// §7.6.1 — single gated manual-command entry for the HMI. Accepts ONLY when this
// Unit is in MANUAL (§3.4) AND the user holds MANUAL access (§7.7). Routes to the
// target module's ManualCommand (through the command surface — defended, not
// bypassed). Logs every accept/reject as a §8.3 event. Concrete Units override
// _M_RouteManual to map TargetPath -> the child module.
METHOD ManualCommandTo : BOOL
VAR_INPUT
    TargetPath : STRING(255);
    Value : DINT;
END_VAR
VAR
    auditSlot : INT;
END_VAR
ManualCommandTo := FALSE;
IF _mode <> E_Mode.MANUAL THEN
    auditSlot := AlarmLog.Raise(Reason := E_Reason.NONE,
        Text := 'std.audit.manualCommandWrongMode', Source := TargetPath,
        Severity := E_Severity.LOW, Category := E_Category.SYSTEM, ResetClass := E_ResetClass.AUTO_RESET);
    IF auditSlot > 0 THEN AlarmLog.Gone(Slot := auditSlot); END_IF
    RETURN;
END_IF
IF NOT Access.PermitsLogged(Gate := E_GatedAction.MANUAL) THEN
    RETURN;                              // §7.7 denial already audited
END_IF
ManualCommandTo := _M_RouteManual(TargetPath := TargetPath, Value := Value);
IF ManualCommandTo THEN
    auditSlot := AlarmLog.Raise(Reason := E_Reason.NONE,
        Text := 'std.audit.manualCommandAccepted', Source := TargetPath,
        Severity := E_Severity.LOW, Category := E_Category.SYSTEM, ResetClass := E_ResetClass.AUTO_RESET);
ELSE
    auditSlot := AlarmLog.Raise(Reason := E_Reason.UNSUPPORTED_COMMAND,
        Text := 'std.audit.manualCommandRejected', Source := TargetPath,
        Severity := E_Severity.LOW, Category := E_Category.SYSTEM, ResetClass := E_ResetClass.AUTO_RESET);
END_IF
IF auditSlot > 0 THEN AlarmLog.Gone(Slot := auditSlot); END_IF
END_METHOD

PROPERTY ModeActive : E_Mode
GET
ModeActive := _mode;
END_GET
END_PROPERTY

PROPERTY ModelCode : STRING(64)
GET
ModelCode := Model.ModelCode;
END_GET
END_PROPERTY

PROPERTY ModuleType : E_ModuleType
GET
ModuleType := E_ModuleType.UNIT;
END_GET
END_PROPERTY

// base first (§3.14.2); then children, one-shot init, mode transition, stall watch
METHOD PROTECTED OnCyclic : DINT
VAR
    publishIdx : INT;
    modeIdx    : E_Mode;
    styleIdx   : E_RunStyle;
    previousMode : E_Mode;
    modeExitResult : DINT;
    highestSeverity : E_Severity;
    alarmActive : BOOL;
    heldReported : BOOL;
END_VAR
OnCyclic := SUPER^.OnCyclic();
_M_SyncModelCatalog();
_M_BeginSequenceScan();                               // §6.10 one-scan result reset for every attached chain
_M_TickChildren();
IF _pLine <> 0 THEN
    IF _lineHost THEN
        _pLine^.Cyclic();                             // §3.8e the hosting root runs the line
    END_IF
    // A line value can change without a write through THIS root: a mirror applies
    // its owner's revision, a second root on the line edits it. Either way this
    // root's manifest now reads differently, so its revision moves.
    IF _pLine^.OutImm.Revision <> _lineRevSeen THEN
        _lineRevSeen := _pLine^.OutImm.Revision;
        ConfigRev := ConfigRev + 1;
    END_IF
END_IF
_M_OeeUpdate();                                       // §8.5.1 time accounting + sampling
M_ShiftTick(Now := F_Now(), Synchronized := F_TimeSynchronized());   // §8.5.2
AlarmLog.Cyclic();                                    // §8.10 shelf auto-expiry
_M_EngineeringCyclic();                               // §7.5.2 standing gate annunciation
_healthPublisher.Cyclic(Input := _healthInput, ParCfg := _healthParCfg,
    Configured := _healthConfigured);                 // §2.7/§8.12 alarm edges + values
SystemHealth := _healthPublisher.Status;
_M_ChartRevCyclic();                                  // §3.13 coalesced chart revision
_M_HeldCyclic();                                      // §7.6.1a hold-to-run re-assert
_M_ConfigPersistCyclic();                             // §3.8b durability window
_M_DrainRestoreLoss();                                // §3.8b restore annunciation
_M_HandleHmiRequest();                                // §3.10 request mailbox
_M_DecisionCyclic();                                  // §6.11 timeout/default/overlap resolver
Access.Cyclic();
alarmActive := _M_HighestSeverity(Highest := highestSeverity);
_towerMapper.Cyclic(MachineState := MachineState, AlarmActive := alarmActive,
    HighestSeverity := highestSeverity,
    OperatorActionRequired := (Decision.Prompt <> ''),
    LampTestRequest := _lampTestRequest, ParCfg := _towerParCfg);
_lampTestRequest := FALSE;
SignalTower := _towerMapper.Status;
// §9.8 data-driven Control On/Off request endpoint. Off wins if both arrive;
// the domain/power-group implementation still validates safety, health and rearm.
ControlOnRequest := FALSE;
ControlOffRequest := FALSE;
IF ReqControlOff THEN
    ReqControlOff := FALSE;
    ReqControlOn := FALSE;
    IF Access.PermitsLogged(Gate := E_GatedAction.POWER_CONTROL) THEN
        ControlOffRequest := TRUE;
    END_IF
ELSIF ReqControlOn THEN
    ReqControlOn := FALSE;
    IF Access.PermitsLogged(Gate := E_GatedAction.POWER_CONTROL) THEN
        ControlOnRequest := TRUE;
    END_IF
END_IF
// §3.14.4 — pending mode change; §3.4.1 style decides graceful vs immediate
IF _modePend THEN
    IF _exec = E_ExecState.BUSY THEN
        IF ModePolicy[TO_INT(_mode)].Style = E_ModeSwitchStyle.GRACEFUL THEN
            _stopReq := TRUE;                             // finish the cycle at its stop point
        ELSE
            modeExitResult := OnModeExit(FirstCall := _modeExitFirst,
                RequestedMode := _modeReq);
            _modeExitFirst := FALSE;
            IF modeExitResult = 0 THEN
                OnAbort();                                // IMMEDIATE: cancel now (override may defer)
            END_IF
        END_IF
    ELSE
        IF _exec <> E_ExecState.READY THEN
            Execute := FALSE;                             // release the run command (§6.1 reset)
        ELSE
            previousMode := _mode;
            _mode := _modeReq;
            _modePend := FALSE;
            _modeExitFirst := FALSE;
            _M_CascadeMode(_mode);                        // §3.7 cascade [TC3]
            OnModeChanged(NewMode := _mode, OldMode := previousMode);
        END_IF
    END_IF
END_IF
// §8.3(c) — automatic fault capture: ERROR entry raises, ERROR exit marks gone
IF (_exec = E_ExecState.ERROR) AND (_faultEvt = 0) THEN
    _faultEvt := AlarmLog.RaiseDiag(D := _diag, ResetClass := E_ResetClass.MANUAL_RESET);
    _M_PartAborted();                  // §3.16.3: a faulted part leaves without a valid result
ELSIF (_exec <> E_ExecState.ERROR) AND (_faultEvt > 0) THEN
    AlarmLog.Gone(Slot := _faultEvt);                            // -> WAIT_RESET (blocking)
    _faultEvt := 0;
END_IF
// §6.9 — instant rollup on awaited Error; adopt a HELD child; stall as PENDING otherwise
IF _exec = E_ExecState.BUSY THEN
    IF (_awaits <> 0) AND_THEN _awaits.FaultActive THEN
        _M_FaultDiag(_awaits.GetFaultSummary());
    ELSE
        // §6.1 HELD — the held module is waiting on a condition it can name, so
        // report THAT instead of letting StallTime expire into a generic stall. A
        // declared wait is not a stall, so the watchdog stays disarmed while it lasts.
        //
        // The hold rolls up whether or not the step awaits the child (§1.1 O1: the
        // project must not have to remember a call to stay correct). `Awaits := 0`
        // says "this step owns the child's FAULT disposition" (§6.9, press AUTO
        // N200 offering scrap/return) - it does not say "stay silent while the ram
        // is HELD". A hold is recoverable information that clears itself and never
        // blocks a restart, so suppressing it only produced a Unit that sat BUSY
        // with an empty diagnostic while its own child correctly reported Held.
        // Prefer the awaited module: when a step named one it is the most specific
        // source. _M_RollupHold is called on exactly the scans the awaited branch
        // did not fire, because TwinCAT does not short-circuit and calling both
        // would let a second held child overwrite the named one.
        heldReported := FALSE;
        IF (_awaits <> 0) AND_THEN _awaits.HoldActive THEN
            _M_HoldDiag(Diag := _awaits.GetFaultSummary());
            heldReported := TRUE;
        ELSE
            heldReported := _M_RollupHold();   // §8.2 first held registered child
        END_IF
        IF heldReported THEN
            _tStall(IN := FALSE);
        ELSE
            IF Held THEN
                _M_ClearPending();     // the hold ended: drop any stall text it outlived
            END_IF
            _tStall(IN := TRUE, PT := SEL(CurrentStep.ExpectedTime > T#0S, StallTime, CurrentStep.ExpectedTime));
            IF _tStall.Q THEN
                _M_StallWalk();
            END_IF
        END_IF
    END_IF
ELSE
    _tStall(IN := FALSE);
END_IF
// §6.9(a) — every new fault joins the shift-change ring, no historian needed
_fTrig(CLK := (_exec = E_ExecState.ERROR));
_errClr(CLK := (_exec <> E_ExecState.ERROR));
IF _errClr.Q THEN
    _M_ResumeSequencesAfterError();   // §6.9 re-evaluate, do not resume blind
END_IF
IF _fTrig.Q THEN
    _M_PushHistory(_diag);
END_IF
// §8.11.4(d) — creeping WORK time is a MAINTENANCE event (Low), not downtime:
// the profiler pulses once per excursion past the configured baseline band.
IF Profiler.DegradedTrig THEN
    _M_RaiseMaintenance(Reason := E_Reason.CYCLE_TIME_DEGRADED,
        Text := 'std.maintenance.cycleTimeDegraded');
END_IF
ModeActivePublished := _mode;
RunningPublished := (_exec = E_ExecState.BUSY);
StopPendingPublished := _stopReq AND (_exec = E_ExecState.BUSY);
FOR publishIdx := 0 TO PL_Fraktal.MODE_COUNT - 1 DO
    modeIdx := publishIdx;
    SupportedModesPublished[publishIdx] := _M_Supports(Mode := modeIdx);
END_FOR
FOR publishIdx := 0 TO 2 DO
    styleIdx := publishIdx;
    SupportedRunStylesPublished[publishIdx] := _M_SupportsRunStyle(Style := styleIdx);
END_FOR
END_METHOD

// §8.13 — derive the tower input from the authoritative active-event table.
METHOD PRIVATE _M_HighestSeverity : BOOL
VAR_IN_OUT
    Highest : E_Severity;
END_VAR
VAR
    i : INT;
END_VAR
_M_HighestSeverity := FALSE;
Highest := E_Severity.LOW;
FOR i := 1 TO PL_Fraktal.MAX_ALARM_ACTIVE DO
    IF AlarmLog.Active[i].State <> E_AlarmState.CLOSED THEN
        IF NOT _M_HighestSeverity OR (AlarmLog.Active[i].Severity > Highest) THEN
            Highest := AlarmLog.Active[i].Severity;
        ELSE
            ;
        END_IF
        _M_HighestSeverity := TRUE;
    ELSE
        ;
    END_IF
END_FOR
END_METHOD

// §8.13 — remote request is MANUAL-gated and starts only while the Unit is idle.
METHOD RequestLampTest : BOOL
RequestLampTest := FALSE;
IF _exec = E_ExecState.BUSY THEN
    RETURN;
END_IF
IF NOT Access.PermitsLogged(Gate := E_GatedAction.MANUAL) THEN
    RETURN;
END_IF
_lampTestRequest := TRUE;
RequestLampTest := TRUE;
END_METHOD

// Startup station-convention seam. Runtime config writes require a registered
// typed capability; this method is not published by OPC UA.
METHOD SetSignalTowerConfig : BOOL
VAR_INPUT
    ParCfg : ST_SignalTowerParCfg;
END_VAR
IF (ParCfg.SchemaVersion <> 1) OR (ParCfg.LampTestDuration <= T#0S) THEN
    SetSignalTowerConfig := FALSE;
    RETURN;
END_IF
_towerParCfg := ParCfg;
SetSignalTowerConfig := TRUE;
END_METHOD

// TC3/platform adapter injection. Raw probe values remain OPC-UA-hidden; the
// health publisher validates and republishes the bounded status surface.
METHOD SetSystemHealth : BOOL
VAR_INPUT
    Input  : ST_SystemHealthInput;
    ParCfg : ST_SystemHealthParCfg;
END_VAR
IF ParCfg.SchemaVersion <> 1 THEN
    SetSystemHealth := FALSE;
    RETURN;
END_IF
_healthInput := Input;
_healthParCfg := ParCfg;
_healthConfigured := TRUE;
SetSystemHealth := TRUE;
END_METHOD

// §3.14 hook — one-shot after first operational scan
METHOD PROTECTED OnInit : DINT
VAR
    i : INT;
END_VAR
OnInit := SUPER^.OnInit();
_M_RestartSequences();         // §6.8 every attached chain starts at N000
SequenceViewEnabled := TRUE;   // §3.13 a Unit has a chain worth drawing;
                               // a concrete Unit may vary this per mode
Access.Setup(Provider := 0, pAlarmLog := ADR(AlarmLog)); // preserves an injected provider
_healthPublisher.Setup(SourcePath := CONCAT(Status.Name, '.SystemHealth'),
    pAlarmLog := ADR(AlarmLog));
// §3.10.2 — seed the manifest revision from boot time so every PLC restart or
// re-activation yields a NEW value (a plain counter would repeat after reboot
// and an HMI could keep a stale manifest undetected). Config writes increment.
ConfigRev := DT_TO_UDINT(F_Now());
// §3.8b — the durability provider defaults to the shipped LOCAL_RETAIN writer.
// SetConfigPersistence may already have replaced it, so this never overwrites an
// injected one.
IF _persistence = 0 THEN
    _persistence := _persistWriter;
END_IF
_liveArmed := TRUE;            // §3.8b the walk is complete: the documents may restore
// The framework's OWN station config is subject to the same rule it imposes on
// every module: version 0 is a first boot that lost nothing, any other
// unrecognized version means a real ModePolicy image was rejected and that is
// annunciated with this root's path. The base used to treat both cases as a
// silent re-initialize, which is exactly the "runs on defaults while presenting
// itself as commissioned" failure §3.8b exists to prevent.
IF NOT M_RestoreStationCfg(pVersion := ADR(_modePolicyVersion),
        SchemaVersion := MODE_POLICY_SCHEMA) THEN
    _M_InitModePolicy();
    FOR i := 0 TO PL_Fraktal.MODE_COUNT - 1 DO
        _modePolicyStored[i] := ModePolicy[i];
    END_FOR
ELSE
    FOR i := 0 TO PL_Fraktal.MODE_COUNT - 1 DO
        ModePolicy[i] := _modePolicyStored[i];
    END_FOR
END_IF
END_METHOD

// §3.14 hook — after the new mode is committed
METHOD PROTECTED OnModeChanged : DINT
VAR_INPUT
    NewMode : E_Mode;
    OldMode : E_Mode;
END_VAR
_M_HostEvent(Kind := E_HostEventKind.MODE_CHANGED, PartUid := '',
    Subject := 'Mode', Value := TO_STRING(TO_DINT(NewMode)),
    Verdict := E_Verdict.NONE, ReasonCode := E_Reason.NONE);
// §3.13 — the chart belongs to the mode that is running. A project writes nothing
// for this: it lands in the base hook every override calls SUPER^ on first (§3.14.2).
_M_ResetSequenceRows();
// §6.8 — and so do the chains: a new mode starts every chain at N000.
_M_RestartSequences();
OnModeChanged := 0;
END_METHOD

// Core §11.6: CHANGEOVER starts when its guided sequence actually starts, not
// merely when the operator selects the mode or transactionally loads a model.
METHOD PROTECTED OnCommandStart : DINT
OnCommandStart := SUPER^.OnCommandStart();
IF _mode = E_Mode.CHANGEOVER THEN
    _M_HostEvent(Kind := E_HostEventKind.CHANGEOVER_STARTED, PartUid := '',
        Subject := 'Model', Value := Model.ModelCode,
        Verdict := E_Verdict.NONE, ReasonCode := E_Reason.NONE);
END_IF
END_METHOD

// §3.14.4 — called every scan while a mode request is pending and the Unit is BUSY.
// Return 0 = consent to immediate cancel (default); >0 = still stopping gracefully.
METHOD PROTECTED OnModeExit : DINT
VAR_INPUT
    FirstCall : BOOL;
    RequestedMode : E_Mode;
END_VAR
OnModeExit := 0;
END_METHOD

// §8.3(b) — deliberate operator reset of blocking events (release-gated per §7.6/§14).
// ONE operator action has to make the Unit restartable, so this closes the blocking
// events AND clears the latched control state they were reporting: see _M_RecoverState.
METHOD OperatorReset : BOOL
IF NOT Access.PermitsLogged(Gate := E_GatedAction.ALARM_RESET) THEN
    OperatorReset := FALSE;            // §7.7
    RETURN;
END_IF
OperatorReset := _M_RecoverState();
OperatorReset := AlarmLog.OperatorReset() OR OperatorReset;
END_METHOD

// §8.3(b)/§6.1 — the control-state half of a reset. Closing the alarm alone left the
// machine locked: the Unit's run command and the child commands its mode chain had
// issued both stayed asserted, and §6.1's Execute-drop reset — the only exit from a
// latched terminal state — needs them LOW. A frozen chain cannot drop them itself,
// because a Unit that is not BUSY never calls _M_Dispatch again, so the step holding
// `child.Execute := TRUE` never runs. Nothing else in the system clears it, and the
// next Start re-issues the same already-TRUE input: no rising edge, the child stays
// in ERROR, and the Unit re-adopts the fault through the §8.2 rollup. That is the
// press hard-lock. Returns TRUE when there was something to recover.
// Deliberately does NOT clear ERROR here: Cyclic keeps that ownership (§6.1), so a
// cause that is still live re-faults on the next command edge instead of vanishing.
METHOD PROTECTED _M_RecoverState : BOOL
_M_RecoverState := FALSE;
IF (_exec <> E_ExecState.ERROR) AND NOT AlarmLog.Blocking THEN
    RETURN;                            // nothing latched: a stray reset changes nothing
END_IF
OnOperatorReset();                     // §3.14 hook: withdraw outputs, reset mode chains
_M_ReleaseChildCommands();             // stranded child commands -> READY next scan
_M_ClearPending();
_stopReq := FALSE;
IF _exec = E_ExecState.BUSY THEN
    // Defined safe reaction (§5.6) for a blocking event raised by application code
    // while the mode chain still runs: a recovery reset cancels what was running
    // rather than leaving a chain we just reset still driving the machine.
    AbortCommand();
END_IF
Execute  := FALSE;                     // stale run command -> Unit READY next scan
_faultEvt := 0;                        // the event is closed here, not by a later Gone()
_M_RecoverState := TRUE;
END_METHOD

// §3.14 hook — an accepted operator reset is recovering this Unit. Override to
// withdraw application outputs and reset application-owned mode chains before the
// base releases the run command; call SUPER^.OnOperatorReset() first (§3.14.2).
// Called only when something was actually latched (ERROR or a blocking alarm), so an
// override may assume it is a recovery, not a routine poll.
METHOD PROTECTED OnOperatorReset : DINT
OnOperatorReset := 0;
END_METHOD

// Application-only seam for an ordinary hardwired fault-reset/acknowledge button,
// mirroring RequestLocalControl (§9.8): it is a METHOD, not OPC UA data, so remote
// clients still go through the access-gated OPERATOR_RESET request and cannot reach
// this path. A cabinet button IS its own authorization (physical presence), so it
// carries no §7.7 session check — but the reset is still audited as a §8.3 event,
// and it recovers exactly the same state as an operator reset, never more.
// The composition root calls this from its hardware driver on the button's rising
// edge, once per root Unit it should clear.
METHOD RequestLocalReset : BOOL
VAR
    auditSlot : INT;
END_VAR
auditSlot := AlarmLog.Raise(Reason := E_Reason.NONE,
    Text := 'std.audit.localResetRequested', Source := _name,
    Severity := E_Severity.LOW, Category := E_Category.SYSTEM,
    ResetClass := E_ResetClass.AUTO_RESET);
IF auditSlot > 0 THEN AlarmLog.Gone(Slot := auditSlot); END_IF
RequestLocalReset := _M_RecoverState();
RequestLocalReset := AlarmLog.OperatorReset() OR RequestLocalReset;
END_METHOD

// §3.8 optional HMI/MES selection catalog. Recipe providers remain pluggable;
// the application registers only the model identities it deliberately exposes.
METHOD RegisterAvailableModel : BOOL
VAR_INPUT
    Id : ST_ModelId;
END_VAR
VAR
    i : INT;
END_VAR
RegisterAvailableModel := FALSE;
IF (Id.ModelCode = '') OR (AvailableModelCount >= PL_Fraktal.MAX_RECIPES) THEN
    RETURN;
END_IF
FOR i := 1 TO AvailableModelCount DO
    IF AvailableModels[i].ModelCode = Id.ModelCode THEN
        RETURN;
    END_IF
END_FOR
AvailableModels[AvailableModelCount + 1] := Id;
AvailableModelCount := AvailableModelCount + 1;
ConfigRev := ConfigRev + 1;    // §3.10.2 — manifest changed
RegisterAvailableModel := TRUE;
END_METHOD

// §9.8 remote control-domain request. The acknowledgement is the result of this
// authorization check; it is never reported accepted before POWER_CONTROL runs.
METHOD RequestControlPower : BOOL
VAR_INPUT
    ControlOn : BOOL;
END_VAR
RequestControlPower := FALSE;
IF NOT Access.PermitsLogged(Gate := E_GatedAction.POWER_CONTROL) THEN
    RETURN;
END_IF
IF ControlOn THEN
    ReqControlOn := TRUE;
    ReqControlOff := FALSE;
ELSE
    ReqControlOff := TRUE;                         // Off wins if both were requested
    ReqControlOn := FALSE;
END_IF
RequestControlPower := TRUE;
END_METHOD

// §6.11 authoritative decision entry. START_STOP is the access gate because the
// answer advances a running Unit chain; option-specific process releases append
// through _M_AppendDecisionInterlocks. A stale/invalid answer never latches.
METHOD SubmitDecision : BOOL
VAR_INPUT
    Option : INT;
END_VAR
VAR_IN_OUT
    Report : ST_ReleaseReport;
END_VAR
Report.Count := 0;
Report.Released := FALSE;
SubmitDecision := FALSE;
IF NOT Access.PermitsLogged(Gate := E_GatedAction.START_STOP) THEN
    _M_AddReason(Report := Report, Text := 'std.release.insufficientStartStop',
        Reason := E_Reason.NONE, Kind := E_ReleaseKind.ACCESS);
END_IF
IF (_exec <> E_ExecState.BUSY) OR (Decision.Prompt = '') THEN
    _M_AddReason(Report := Report, Text := 'std.release.noActiveDecision',
        Reason := E_Reason.NONE, Kind := E_ReleaseKind.OTHER);
ELSIF (Option < 1) OR (Option > PL_Fraktal.MAX_OPTIONS) THEN
    _M_AddReason(Report := Report, Text := 'std.release.invalidDecisionOption',
        Reason := E_Reason.UNSUPPORTED_COMMAND, Kind := E_ReleaseKind.OTHER);
ELSIF Decision.Options[Option] = '' THEN
    _M_AddReason(Report := Report, Text := 'std.release.invalidDecisionOption',
        Reason := E_Reason.UNSUPPORTED_COMMAND, Kind := E_ReleaseKind.OTHER);
ELSE
    _M_AppendDecisionInterlocks(Option := Option, Report := Report);
END_IF
Report.Released := (Report.Count = 0);
IF Report.Released THEN
    DecisionAnswer := Option;
    SubmitDecision := TRUE;
END_IF
END_METHOD

// §7.7 persistent per-root policy edit. The policy's own ACCESS_POLICY threshold
// is rechecked before any threshold — including itself — can change.
METHOD SetAccessLevel : BOOL
VAR_INPUT
    Gate : E_GatedAction;
    Level : E_AccessLevel;
END_VAR
SetAccessLevel := FALSE;
IF NOT Access.PermitsLogged(Gate := E_GatedAction.ACCESS_POLICY) THEN
    RETURN;
END_IF
// Never allow an anonymous/lower session to raise the policy above itself and
// strand the retained station configuration without a usable administrator.
IF (Gate = E_GatedAction.ACCESS_POLICY) AND (Level > Access.CurrentLevel) THEN
    RETURN;
END_IF
SetAccessLevel := Access.ConfigureRequired(Gate := Gate, Level := Level);
IF SetAccessLevel THEN
    ConfigRev := ConfigRev + 1;
END_IF
END_METHOD

// §7.7 persistent idle timeout (0 = never), self-gated by ACCESS_POLICY.
METHOD SetSessionTimeout : BOOL
VAR_INPUT
    TimeoutMs : UDINT;
END_VAR
SetSessionTimeout := FALSE;
IF NOT Access.PermitsLogged(Gate := E_GatedAction.ACCESS_POLICY) THEN
    RETURN;
END_IF
SetSessionTimeout := Access.ConfigureSessionTimeout(TimeoutMs := TimeoutMs);
IF SetSessionTimeout THEN
    ConfigRev := ConfigRev + 1;
END_IF
END_METHOD

// §3.8a/§7.7 centralized HMI configuration authority. Concrete overrides never
// need to remember DATA_WRITE or root ownership; they validate only their field.
METHOD WriteConfig : BOOL
VAR_INPUT
    TargetPath : STRING(255);
    WriteKey : STRING(160);
    Revision : DINT;
    TextValue : STRING(255);
END_VAR
WriteConfig := FALSE;
IF NOT _M_ConfigRestored() THEN
    RETURN;                            // §3.8b the restore would replay over it
END_IF
IF (WriteKey = '') OR (Revision <= 0)
OR NOT _M_OwnsModulePath(Path := TargetPath) THEN
    RETURN;
END_IF
// §3.8d - the VALUE's effective write level (its class, raised by its own
// minimum); DATA_WRITE for a value in the built-in class, as before.
IF NOT Access.M_PermitsLevelLogged(Required := _M_DataLevelOf(TargetPath := TargetPath,
        WriteKey := WriteKey, ForWrite := TRUE)) THEN
    RETURN;
END_IF
WriteConfig := _M_WriteBaseConfig(TargetPath := TargetPath, WriteKey := WriteKey,
    Revision := TO_UDINT(Revision), TextValue := TextValue, Commit := TRUE);
IF NOT WriteConfig THEN
    WriteConfig := _M_RouteConfigWrite(TargetPath := TargetPath,
        WriteKey := WriteKey, Revision := TO_UDINT(Revision), TextValue := TextValue);
END_IF
// §3.8a - a model-data value lives in a recipe record too. Another model's edit
// exists ONLY in that record, so failing to save it fails the write; the active
// model's edit is already live, and saving it keeps it across a changeover.
IF WriteConfig AND (TargetPath = Status.Name) AND _M_ModelScopedKey(WriteKey := WriteKey) THEN
    IF NOT _M_SaveModelData() AND (_pModelView <> 0) THEN
        WriteConfig := FALSE;
    END_IF
END_IF
IF WriteConfig THEN
    ConfigRev := ConfigRev + 1;
    _M_MarkPersistPending();           // §3.8b: accepted is LIVE, not yet DURABLE
END_IF
END_METHOD

// §3.8c - the root authority for a capture. Deliberately the same gate, the same
// ownership check and the same ConfigRev bump as WriteConfig: a capture is a
// write whose value came from the machine, and it is no more and no less
// privileged than one the operator typed (§3.8c(d)).
METHOD CaptureConfig : BOOL
VAR_INPUT
    TargetPath : STRING(255);
    WriteKey   : STRING(160);
    Revision   : DINT;
END_VAR
CaptureConfig := FALSE;
IF NOT _M_ConfigRestored() THEN
    RETURN;
END_IF
IF (WriteKey = '') OR (Revision <= 0)
OR NOT _M_OwnsModulePath(Path := TargetPath) THEN
    RETURN;
END_IF
IF NOT Access.M_PermitsLevelLogged(Required := _M_DataLevelOf(TargetPath := TargetPath,
        WriteKey := WriteKey, ForWrite := TRUE)) THEN
    RETURN;
END_IF
// Framework-owned keys offer no capture: they are policy, not measurements.
CaptureConfig := M_ApplyCapture(Scope := TargetPath, WriteKey := WriteKey,
    Revision := TO_UDINT(Revision), RootReady := (_exec = E_ExecState.READY));
IF CaptureConfig THEN
    ConfigRev := ConfigRev + 1;
END_IF
END_METHOD

// Core §7.5.1 — inject the station's commissioning/engineering gate register at
// Setup, the same shape as SetPartCarrier. Wiring it is what makes the §7.5.2
// standing annunciation appear and what arms the §10.5.1 force surface; a Unit
// with no register is a production Unit and both are simply absent.
//
// Declaring the framework's OWN force gate happens here rather than in the
// project, so a composition root that wires the register cannot forget it
// (§1.1 O1) and cannot arm forcing without also annunciating it.
METHOD SetEngineeringMode
VAR_INPUT
    Mode : REFERENCE TO FB_EngineeringMode;
END_VAR
_engineering REF= Mode;
IF __ISVALIDREF(_engineering) THEN
    _engineering.M_DeclareOutputForcing();
ELSE
    ;
END_IF
END_METHOD

// Core §10.5.1 rules 1 and 3 — may a held force set-point be applied to this
// Unit's outputs right now? The project hardware driver passes the result to
// FB_IoTopologyPublisher.M_ApplyForces every scan, and ForceChannel gates the
// operator request on the identical predicate, so "accepted" and "applied" can
// never disagree. Everything else about a force (access, ownership, direction,
// mapping) is proved elsewhere; this is only the build gate and the mode/state.
METHOD M_ForcePermitted : BOOL
M_ForcePermitted := FALSE;
IF NOT __ISVALIDREF(_engineering) THEN
    RETURN;
END_IF
IF NOT _engineering.ForcingActive THEN
    RETURN;
END_IF
// A running module reasserts its own outputs, so a force is only honest while
// the Unit is idle in MANUAL; leaving either withdraws every force (§10.5.1(3)).
M_ForcePermitted := (_mode = E_Mode.MANUAL) AND (_exec = E_ExecState.READY);
END_METHOD

// Core §7.5.2 — the standing annunciation: one LOW/SYSTEM/AUTO_RESET event per
// registered gate, for as long as that gate is registered.
//
// Why each choice is the way it is, because every one of them is load-bearing:
//   AUTO_RESET  a MANUAL_RESET event refuses Start (§8.3(b)), which would make
//               commissioning gates block the commissioning they exist to serve;
//   LOW/SYSTEM  the lowest priority and the lowest risk class - this says how the
//               software was BUILT, not that the process or safety is impaired,
//               and a louder class would displace real alarms (§8.9);
//   unclearable OperatorReset only closes MANUAL_RESET events, so no operator
//               action reaches this one, and its §8.9 record is not shelvable, so
//               §8.10 cannot silence it either. It closes when the gate is gone -
//               which, gates being build constants, means a new download.
METHOD PRIVATE _M_EngineeringCyclic
VAR
    i : INT;
    gateCount : INT;
END_VAR
IF NOT __ISVALIDREF(_engineering) THEN
    RETURN;
END_IF
gateCount := _engineering.Count;
IF gateCount > PL_Fraktal.MAX_ENGINEERING_GATES THEN
    gateCount := PL_Fraktal.MAX_ENGINEERING_GATES;
END_IF
FOR i := 1 TO gateCount DO
    // Self-healing on purpose. If this slot were ever closed and reused by
    // another event, a remembered index would leave the annunciation silently
    // absent for the rest of the run - the one failure mode a non-clearable
    // message must not have. Re-verify identity, then re-raise.
    IF _engineeringEvt[i] > 0 THEN
        IF (AlarmLog.Active[_engineeringEvt[i]].State = E_AlarmState.CLOSED)
        OR (AlarmLog.Active[_engineeringEvt[i]].ReasonCode <> E_Reason.COMMISSIONING_GATE_ACTIVE) THEN
            _engineeringEvt[i] := 0;
        ELSE
            ;
        END_IF
    ELSE
        ;
    END_IF
    IF _engineeringEvt[i] = 0 THEN
        _engineeringEvt[i] := AlarmLog.Raise(Reason := E_Reason.COMMISSIONING_GATE_ACTIVE,
            Text := _engineering.Gates[i].DescriptionKey, Source := _name,
            Severity := E_Severity.LOW, Category := E_Category.SYSTEM,
            ResetClass := E_ResetClass.AUTO_RESET);
    ELSE
        ;
    END_IF
END_FOR
END_METHOD

// §10.5.1 centralized force authority. Only an idle MANUAL Unit may reach the
// application resolver; that resolver still proves root ownership, OUTPUT,
// non-safety identity, mapping and the channel-specific release.
METHOD ForceChannel : BOOL
VAR_INPUT
    ChannelPath : STRING(255);
    Force : BOOL;
    BoolText : STRING(255);
    AnalogText : STRING(160);
END_VAR
ForceChannel := FALSE;
IF NOT Access.PermitsLogged(Gate := E_GatedAction.MANUAL) THEN
    RETURN;
END_IF
// §10.5.1 rules 1 and 3 in one predicate, the same one the hardware driver
// applies each scan - so the request can never be accepted under conditions
// under which the force would not actually be applied.
IF NOT M_ForcePermitted() OR (ChannelPath = '') THEN
    RETURN;
END_IF
ForceChannel := _M_RouteForceChannel(ChannelPath := ChannelPath, Force := Force,
    BoolText := BoolText, AnalogText := AnalogText);
END_METHOD

// Core §7.8 — full rollup for the simpler gated Unit actions (Stop, ALARM_RESET,
// CHANGEOVER, MODE_CHANGE, step). Same predicate the gates use. Start has its own
// richer ReleaseReportStart (interlocks); manual has ReleaseReportManual (target).
METHOD ReleaseReportAction : BOOL
VAR_INPUT
    Gate : E_GatedAction;
END_VAR
VAR_IN_OUT
    Report : ST_ReleaseReport;
END_VAR
Report.Count := 0;
Report.Released := FALSE;
// access is the common gate
IF NOT Access.Permits(Gate := Gate) THEN
    _M_AddReason(Report := Report, Text := 'std.release.insufficientAction', Reason := E_Reason.NONE, Kind := E_ReleaseKind.ACCESS);
END_IF
// per-action state preconditions
CASE Gate OF
    E_GatedAction.CHANGEOVER:
        IF _exec = E_ExecState.BUSY THEN
            _M_AddReason(Report := Report, Text := 'std.release.changeoverRunning', Reason := E_Reason.NONE, Kind := E_ReleaseKind.MODE);
        END_IF
    E_GatedAction.ALARM_RESET:
        IF NOT AlarmLog.Blocking THEN
            _M_AddReason(Report := Report, Text := 'std.release.noBlockingAlarm', Reason := E_Reason.NONE, Kind := E_ReleaseKind.OTHER);
        END_IF
    E_GatedAction.MODE_CHANGE:
        IF _modePend THEN
            _M_AddReason(Report := Report, Text := 'std.release.modeChangeAlreadyPending', Reason := E_Reason.NONE, Kind := E_ReleaseKind.MODE);
        ELSIF (_exec = E_ExecState.BUSY)
        AND (ModePolicy[TO_INT(_mode)].Shield = E_ModeSwitchShield.BLOCKED_WHILE_RUNNING) THEN
            _M_AddReason(Report := Report, Text := 'std.release.modeSwitchBlockedWhileRunning',
                Reason := E_Reason.NONE, Kind := E_ReleaseKind.MODE);
        ELSE
            ;
        END_IF
ELSE
    ;                                          // actions with no extra state predicate
END_CASE
Report.Released := (Report.Count = 0);
ReleaseReportAction := Report.Released;
END_METHOD

// Core §7.8 — full rollup of why a manual command to Target would be refused (§7.6.1).
METHOD ReleaseReportManual : BOOL
VAR_INPUT
    TargetPath : STRING(255);
    Value : DINT;
END_VAR
VAR_IN_OUT
    Report : ST_ReleaseReport;
END_VAR
Report.Count := 0;
Report.Released := FALSE;
IF _mode <> E_Mode.MANUAL THEN
    _M_AddReason(Report := Report, Text := 'std.release.manualModeRequired', Reason := E_Reason.NONE, Kind := E_ReleaseKind.MODE);
END_IF
IF NOT Access.Permits(Gate := E_GatedAction.MANUAL) THEN
    _M_AddReason(Report := Report, Text := 'std.release.insufficientManual', Reason := E_Reason.NONE, Kind := E_ReleaseKind.ACCESS);
END_IF
_M_AppendManualInterlocks(TargetPath := TargetPath, Value := Value, Report := Report);  // §7.6, target+command-aware
Report.Released := (Report.Count = 0);
ReleaseReportManual := Report.Released;
END_METHOD

// Core §7.8 — pure query: the FULL rollup of why Start would be refused right now.
// This is the authoritative machine predicate consumed by Start (no drift).
// Released = TRUE means Start proceeds. Lists mode + access + blocking-alarm,
// control-domain, and concrete mode-entry release reasons. The caller owns the
// bounded report storage; returning this large record by value can overflow a
// TwinCAT task stack when Start consumes the result.
METHOD ReleaseReportStart : BOOL
VAR_IN_OUT
    Report : ST_ReleaseReport;
END_VAR
Report.Count := 0;
Report.Released := FALSE;
// access (§7.7)
IF NOT Access.Permits(Gate := E_GatedAction.START_STOP) THEN
    _M_AddReason(Report := Report, Text := 'std.release.insufficientStartStop', Reason := E_Reason.NONE, Kind := E_ReleaseKind.ACCESS);
END_IF
// mode / run state (§3.4)
IF _modePend THEN
    _M_AddReason(Report := Report, Text := 'std.release.modeChangePending', Reason := E_Reason.NONE, Kind := E_ReleaseKind.MODE);
END_IF
IF _mode = E_Mode.MANUAL THEN
    _M_AddReason(Report := Report, Text := 'std.release.manualHasNoAutoSequence', Reason := E_Reason.NONE, Kind := E_ReleaseKind.MODE);
END_IF
IF _exec <> E_ExecState.READY THEN
    _M_AddReason(Report := Report, Text := 'std.release.unitNotReady', Reason := E_Reason.NONE, Kind := E_ReleaseKind.MODE);
END_IF
// blocking alarm (§8.3)
IF AlarmLog.Blocking THEN
    _M_AddReason(Report := Report, Text := 'std.release.manualReset', Reason := E_Reason.NONE, Kind := E_ReleaseKind.ALARM);
END_IF
// lost configuration image (§3.8b): the DEPLOYMENT's declared consequence. The
// policy was stored and published but read nowhere, so a station that declared
// BLOCK_UNTIL_ACKNOWLEDGED started on defaults anyway. This is where it is read.
IF ConfigPersist.RestoreLost AND NOT ConfigPersist.RestoreAcknowledged
AND (ConfigPersist.RestorePolicy = E_ConfigRestorePolicy.BLOCK_UNTIL_ACKNOWLEDGED) THEN
    _M_AddReason(Report := Report, Text := 'std.release.configRestoreUnacknowledged', Reason := E_Reason.CONFIG_RESTORE_LOST, Kind := E_ReleaseKind.ALARM);
END_IF
// §3.8b - the live documents are still being read back: the running values are
// not yet the ones last made durable.
IF NOT _M_ConfigRestored() THEN
    _M_AddReason(Report := Report, Text := 'std.release.configRestoring', Reason := E_Reason.NONE, Kind := E_ReleaseKind.OTHER);
END_IF
IF ControlDomain.Present AND NOT ControlDomain.ReadyForStart THEN
    _M_AddReason(Report := Report, Text := 'std.release.controlDomainNotReady', Reason := E_Reason.NONE, Kind := E_ReleaseKind.INTERLOCK);
END_IF
// active mode's immediate entry/frontier conditions (concrete override)
_M_AppendInterlocks(Report := Report);
Report.Released := (Report.Count = 0);
ReleaseReportStart := Report.Released;
END_METHOD

// §8.5.1 — clear accumulators + ring (shift start). Gated: §7.7 DATA_WRITE; audited §8.3.
METHOD ResetOee : BOOL
VAR
    i : INT;
    auditSlot : INT;
END_VAR
IF NOT Access.PermitsLogged(Gate := E_GatedAction.DATA_WRITE) THEN
    ResetOee := FALSE;
    RETURN;
END_IF
_oeeGoodBase := GoodCount;
_oeeNokBase := NokCount;
Oee.RunMs := 0; Oee.DownMs := 0; Oee.IdleMs := 0;
FOR i := 1 TO PL_Fraktal.MAX_OEE_SAMPLES DO
    OeeTrend[i].Oee := 0.0; OeeTrend[i].OeeValid := FALSE;
    OeeTrend[i].Availability := 0.0; OeeTrend[i].Performance := 0.0; OeeTrend[i].Quality := 0.0;
END_FOR
OeeTrendHead := 0;
_oeeSampMs := 0;
_M_OeeCompute();
_shiftManualReset := TRUE;                  // §8.5.2(c): the shift record will say so
auditSlot := AlarmLog.Raise(Reason := E_Reason.NONE,
    Text := 'std.audit.oeeReset', Source := _name,
    Severity := E_Severity.LOW, Category := E_Category.SYSTEM, ResetClass := E_ResetClass.AUTO_RESET);
IF auditSlot > 0 THEN AlarmLog.Gone(Slot := auditSlot); END_IF
ResetOee := TRUE;
END_METHOD

// §3.4.2 — HMI HOLD_TO_RUN input. NON-SAFETY (§9): never a dead-man; interlocks
// still apply at every step. TRUE only while the operator holds the button.
METHOD SetHoldRun : BOOL
VAR_INPUT
    Held : BOOL;
END_VAR
IF Held AND (NOT Access.PermitsLogged(Gate := E_GatedAction.START_STOP)
OR (RunStyle <> E_RunStyle.HOLD_TO_RUN) OR (_exec <> E_ExecState.BUSY)) THEN
    SetHoldRun := FALSE;
    RETURN;
END_IF
_holdRun := Held;                     // FALSE is always accepted so a hold cannot stick
SetHoldRun := TRUE;
END_METHOD

// §8.5.1 — configure the ideal cycle time (per model, §3.8). 0 disables Performance.
METHOD SetIdealCycle : BOOL
VAR_INPUT
    Ms : UDINT;
END_VAR
Oee.IdealCycleMs := Ms;
SetIdealCycle := TRUE;
END_METHOD

// §3.4/§3.7 — FALSE = unsupported (graceful rejection); TRUE = committed or pending
METHOD SetMode : BOOL
VAR_INPUT
    Mode : E_Mode;
END_VAR
IF NOT Access.PermitsLogged(Gate := E_GatedAction.MODE_CHANGE) THEN
    SetMode := FALSE;                  // §7.7(c): who-gate ANDs the machine gates
    RETURN;
END_IF
IF NOT _M_Supports(Mode) THEN
    SetMode := FALSE;
    RETURN;
END_IF
IF (Mode = _mode) AND NOT _modePend THEN
    SetMode := TRUE;
    RETURN;
END_IF
// §3.4.1 shield: policy of the mode being LEFT governs while its sequence runs
IF (_exec = E_ExecState.BUSY)
AND (ModePolicy[TO_INT(_mode)].Shield = E_ModeSwitchShield.BLOCKED_WHILE_RUNNING) THEN
    SetMode := FALSE;                  // must Stop first (graceful rejection, not a fault)
    RETURN;
END_IF
IF (NOT _modePend) OR (_modeReq <> Mode) THEN
    _modeExitFirst := TRUE;
END_IF
_modeReq := Mode;
_modePend := TRUE;
SetMode := TRUE;
END_METHOD

// §3.1b/§3.8 — transactional model change: prepare the whole subtree, then commit.
METHOD SetModel : BOOL
VAR_INPUT
    Id : ST_ModelId;
END_VAR
IF NOT Access.PermitsLogged(Gate := E_GatedAction.CHANGEOVER) THEN
    SetModel := FALSE;                 // §7.7
    RETURN;
END_IF
IF _exec = E_ExecState.BUSY THEN
    SetModel := FALSE;                 // changeover is not mid-cycle (§3.8 loads at CHANGEOVER)
    RETURN;
END_IF
IF NOT PrepareRecipe(Model := Id) THEN
    AbortRecipe();
    SetModel := FALSE;
    RETURN;
END_IF
CommitRecipe();                         // infallible after successful preparation
Model := Id;                           // identity changes only after subtree commit
ConfigRev := ConfigRev + 1;            // §3.10.2 — recipe/config leaves changed
SetModel := TRUE;
END_METHOD

// §11.6.1 internal composition seam; not a remote command surface.
METHOD M_PublishMaterialChanged : BOOL
VAR_INPUT
    Material : STRING(80);
    Value    : STRING(80);
END_VAR
M_PublishMaterialChanged := _M_HostEvent(
    Kind := E_HostEventKind.MATERIAL_CHANGED, PartUid := '', Subject := Material,
    Value := Value, Verdict := E_Verdict.NONE, ReasonCode := E_Reason.NONE);
END_METHOD

// §11.6.1 internal composition seam; not a remote command surface.
METHOD M_PublishToolChanged : BOOL
VAR_INPUT
    Tool  : STRING(80);
    Value : STRING(80);
END_VAR
M_PublishToolChanged := _M_HostEvent(
    Kind := E_HostEventKind.TOOL_CHANGED, PartUid := '', Subject := Tool,
    Value := Value, Verdict := E_Verdict.NONE, ReasonCode := E_Reason.NONE);
END_METHOD

// §11.6.2 inject an optional OPC UA/MES/REST/MQTT delivery adapter.
METHOD M_SetHostEventSink : BOOL
VAR_INPUT
    Sink : I_HostEventSink;
END_VAR
M_SetHostEventSink := HostEvents.SetSink(Sink := Sink);
END_METHOD

// §3.16.2 — inject the part carrier at the composition root (0 = traceability off).
// Source-agnostic: BY_POSITION local, RFID, DataMatrix, or host, behind I_PartCarrier.
METHOD SetPartCarrier : BOOL
VAR_INPUT
    Carrier : I_PartCarrier;
END_VAR
_carrier := Carrier;
SetPartCarrier := (Carrier <> 0);
END_METHOD

// §3.4.2 — HMI selects the run style for the active mode. Modes that don't opt in
// (see _M_SupportsRunStyle) reject non-CONTINUOUS. Access: MODE_CHANGE-gated (§7.7).
METHOD SetRunStyle : BOOL
VAR_INPUT
    Style : E_RunStyle;
END_VAR
IF NOT Access.PermitsLogged(Gate := E_GatedAction.MODE_CHANGE) THEN
    SetRunStyle := FALSE;
    RETURN;
END_IF
IF (Style <> E_RunStyle.CONTINUOUS) AND NOT _M_SupportsRunStyle(Style := Style) THEN
    SetRunStyle := FALSE;               // mode didn't opt into stepping (graceful reject)
    RETURN;
END_IF
RunStyle := Style;
SetRunStyle := TRUE;
END_METHOD

// §8.10 — gated HMI entry: shelve an active alarm's ANNUNCIATION (control untouched).
// §7.7 ALARM_SHELVE + audit; refuses SAFETY / unrationalized reasons (AlarmLog rules).
METHOD ShelveAlarm : BOOL
VAR_INPUT
    Slot      : INT;
    DurationS : UDINT;
END_VAR
IF NOT Access.PermitsLogged(Gate := E_GatedAction.ALARM_SHELVE) THEN
    ShelveAlarm := FALSE;
    RETURN;
END_IF
ShelveAlarm := AlarmLog.Shelve(Slot := Slot, DurationS := DurationS);
END_METHOD

// §3.3/§6 intro — the run IS a §6.1 command.
// §7.8: ReleaseReportStart is the authoritative machine gate as well as the
// operator explanation, so a concrete Unit cannot report an interlock it ignores.
// Build directly into the published response storage: ST_ReleaseReport is too
// large for nested by-value/local copies on a small TwinCAT task stack.
METHOD Start : BOOL
IF NOT Access.PermitsLogged(Gate := E_GatedAction.START_STOP) THEN
    Start := FALSE;                    // §7.7
    RETURN;
END_IF
IF ReleaseReportStart(Report := HmiResponse.Report) THEN
    _stopReq := FALSE;                 // §8.3(b): a MANUAL_RESET event blocks restart
    Execute := TRUE;
    Start := TRUE;
ELSE
    Start := FALSE;
END_IF
END_METHOD

// §3.4.2 — HMI single-step: request advance of one step (edge-consumed by _M_StepGate).
METHOD StepRequest : BOOL
IF NOT Access.PermitsLogged(Gate := E_GatedAction.START_STOP)
OR (RunStyle <> E_RunStyle.SINGLE_STEP) OR (_exec <> E_ExecState.BUSY) THEN
    StepRequest := FALSE;
    RETURN;
END_IF
_stepReq := TRUE;
StepRequest := TRUE;
END_METHOD

// §3.3 — stop after the current cycle
METHOD Stop : BOOL
IF NOT Access.PermitsLogged(Gate := E_GatedAction.START_STOP) THEN
    Stop := FALSE;                     // §7.7
    RETURN;
END_IF
IF _exec = E_ExecState.BUSY THEN
    _stopReq := TRUE;
ELSE
    _stopReq := FALSE;
    Execute := FALSE;                  // release a terminal run command (ERROR/DONE/ABORTED)
END_IF
Stop := TRUE;
END_METHOD

// §3.4 — TRUE while a stop is requested but the sequence is still finishing
// (running -> stopping). HMI blinks the stop button on this.
PROPERTY StopPending : BOOL
GET
StopPending := _stopReq AND (_exec = E_ExecState.BUSY);
END_GET
END_PROPERTY

// §8.10 — gated HMI entry: restore annunciation.
METHOD UnshelveAlarm : BOOL
VAR_INPUT
    Slot : INT;
END_VAR
IF NOT Access.PermitsLogged(Gate := E_GatedAction.ALARM_SHELVE) THEN
    UnshelveAlarm := FALSE;
    RETURN;
END_IF
UnshelveAlarm := AlarmLog.Unshelve(Slot := Slot);
END_METHOD

METHOD PRIVATE _M_SyncModelCatalog
VAR
    i : INT;
    j : INT;
    id : ST_ModelId;
    exists : BOOL;
    found : UINT;
    info : ST_ConfigSetInfo;
    record : ST_ConfigRecord;
END_VAR
IF _modelCatalog = 0 THEN ModelCapacity := 0; RETURN; END_IF
IF _modelCatalogSeen = _modelCatalog.M_ModelCount(RecipeKey := _modelKey) THEN RETURN; END_IF
_modelCatalogSeen := _modelCatalog.M_ModelCount(RecipeKey := _modelKey);
FOR i := 1 TO _modelCatalog.M_ModelCount(RecipeKey := _modelKey) DO
    IF _modelCatalog.M_ModelAt(RecipeKey := _modelKey, Index := i, Id := id) THEN
        exists := FALSE;
        FOR j := 1 TO AvailableModelCount DO
            IF AvailableModels[j].ModelCode = id.ModelCode THEN exists := TRUE; END_IF
        END_FOR
        IF NOT exists THEN RegisterAvailableModel(Id := id); END_IF
    END_IF
END_FOR
ModelCapacity := _modelCatalog.M_ModelCapacity(RecipeKey := _modelKey);
IF ModelCapacity > PL_Fraktal.MAX_RECIPES THEN ModelCapacity := PL_Fraktal.MAX_RECIPES; END_IF
IF _modelCatalog.M_TakeCatalogRestoreLoss(Found => found) THEN
    _restoreLost := TRUE;
    _restoreFound := found;
    _restoreExpected := 1;
END_IF
IF NOT _M_CaptureConfig(SetName := '_validation', Kind := E_ConfigKind.PAR_CFG, ModelIndex := 0) THEN
    ModelCapacity := 0; RETURN;
END_IF
_snapshot.M_ReadInfo(SetName := '_validation', Info := info);
FOR i := 1 TO info.RecordCount DO
    _snapshot.M_ReadRecord(SetName := '_validation', Index := i, Record := record);
    IF NOT _M_OwnsModelRecord(Record := record) THEN ModelCapacity := 0; EXIT; END_IF
END_FOR
END_METHOD

METHOD PRIVATE _M_OwnsModelRecord : BOOL
VAR_INPUT
    Record : ST_ConfigRecord;
END_VAR
VAR
    i : INT;
END_VAR
_M_OwnsModelRecord := FALSE;
IF (Record.Scope <> Status.Name) OR (Record.Kind <> E_ConfigKind.PAR_CFG) THEN RETURN; END_IF
FOR i := 1 TO _nConfigWrite DO
    IF _pConfigWrite[i - 1].Key = Record.WriteKey THEN
        _M_OwnsModelRecord := (_pConfigWrite[i - 1].Kind = E_ConfigKind.PAR_CFG)
            AND (_pConfigWrite[i - 1].pTarget >= _pModelRegion)
            AND (_pConfigWrite[i - 1].pTarget < _pModelRegion + _modelRegionSize);
        RETURN;
    END_IF
END_FOR
END_METHOD

// Freeze untrusted storage before validation or a commit pass.
METHOD PRIVATE _M_CopySet : BOOL
VAR_INPUT
    SetName : STRING(80);
END_VAR
VAR
    info : ST_ConfigSetInfo;
    record : ST_ConfigRecord;
    i : INT;
END_VAR
_M_CopySet := FALSE;
_exportNext := 0;
IF _configStore = 0 THEN RETURN; END_IF
IF NOT _configStore.M_ReadInfo(SetName := SetName, Info := info) THEN RETURN; END_IF
IF (info.SetName <> SetName) OR (info.RecordCount < 1)
OR (info.RecordCount > PL_Fraktal.MAX_SET_RECORDS) THEN RETURN; END_IF
IF NOT _loadSnapshot.M_SaveBegin(Info := info) THEN RETURN; END_IF
FOR i := 1 TO info.RecordCount DO
    IF NOT _configStore.M_ReadRecord(SetName := SetName, Index := i, Record := record) THEN
        _loadSnapshot.M_SaveAbort(); RETURN;
    END_IF
    IF NOT _loadSnapshot.M_SaveRecord(Record := record) THEN
        _loadSnapshot.M_SaveAbort(); RETURN;
    END_IF
END_FOR
_M_CopySet := _loadSnapshot.M_SaveCommit();
END_METHOD

// Reuse the capability walk for immutable export and complete-set validation.
METHOD PRIVATE _M_CaptureConfig : BOOL
VAR_INPUT
    SetName : STRING(80);
    Kind : E_ConfigKind;
    ModelIndex : UDINT;
END_VAR
_exportNext := 0; // every replacement invalidates the old immutable cursor
_M_CaptureConfig := _M_CaptureInto(Store := _snapshot, SetName := SetName, Kind := Kind,
    ModelIndex := ModelIndex);
END_METHOD

// The capability walk as one set in Store. The live documents capture into
// _loadSnapshot, so writing them never invalidates an export of _snapshot.
METHOD PRIVATE _M_CaptureInto : BOOL
VAR_INPUT
    Store : I_ConfigStore;
    SetName : STRING(80);
    Kind : E_ConfigKind;
    ModelIndex : UDINT;
END_VAR
VAR
    info : ST_ConfigSetInfo;
    records : INT;
END_VAR
_M_CaptureInto := FALSE;
IF NOT _M_OpenModelView(Index := ModelIndex) THEN RETURN; END_IF
info.SetName := SetName;
info.Used := TRUE;
info.RootIdentity := Status.Name;
info.SetSchema := CONFIG_SET_SCHEMA;
info.ConfigRev := ConfigRev;
info.Kind := Kind;
info.ModelCode := Model.ModelCode;
IF ModelIndex > 0 THEN info.ModelCode := AvailableModels[ModelIndex].ModelCode; END_IF
IF Kind <> E_ConfigKind.PAR_CFG THEN info.ModelCode := ''; END_IF
info.CreatedAt := F_Now();
info.TimeSynchronized := F_TimeSynchronized();
IF _configPager.M_SetupSetSave(Store := Store, Info := info) THEN
    M_AppendConfig(Pager := _configPager);
    _M_CaptureInto := _configPager.M_FinishSetSave(Records => records);
END_IF
_pModelView := 0;
END_METHOD

// Exact current capability identity/type/revision; no blanket stale migration.
// AnyRevision: a restored document carries the ConfigRev of an earlier run, which
// says nothing about this one; the per-record identity, type and revision still do.
METHOD PRIVATE _M_ValidateSetShape : BOOL
VAR_INPUT
    Store : I_ConfigStore;
    Info : ST_ConfigSetInfo;
    AnyRevision : BOOL;
END_VAR
VAR
    expectedInfo : ST_ConfigSetInfo;
    expected : ST_ConfigRecord;
    record : ST_ConfigRecord;
    i : INT;
    j : INT;
    hits : INT;
END_VAR
_M_ValidateSetShape := FALSE;
IF (Store = 0) OR (Info.RootIdentity <> Status.Name)
OR (Info.SetSchema <> CONFIG_SET_SCHEMA)
OR (Info.RecordCount < 1) OR (Info.RecordCount > PL_Fraktal.MAX_SET_RECORDS) THEN
    _M_RejectConfigSet(Scope := Info.RootIdentity, Key := Info.SetName); RETURN;
END_IF
IF NOT AnyRevision AND ((Info.ConfigRev = 0) OR (Info.ConfigRev > ConfigRev)) THEN
    _M_RejectConfigSet(Scope := Info.RootIdentity, Key := Info.SetName); RETURN;
END_IF
IF NOT _snapshot.M_ReadInfo(SetName := '_validation', Info := expectedInfo) THEN RETURN; END_IF

FOR i := 1 TO Info.RecordCount DO
    IF NOT Store.M_ReadRecord(SetName := Info.SetName, Index := i, Record := record) THEN RETURN; END_IF
    hits := 0;
    FOR j := 1 TO expectedInfo.RecordCount DO
        _snapshot.M_ReadRecord(SetName := '_validation', Index := j, Record := expected);
        IF (record.Scope = expected.Scope) AND (record.WriteKey = expected.WriteKey) THEN
            IF (record.Kind <> expected.Kind) OR (record.ValueType <> expected.ValueType)
            OR (record.Revision <> expected.Revision) THEN
                _M_RejectConfigSet(Scope := record.Scope, Key := record.WriteKey); RETURN;
            END_IF
            hits := hits + 1;
        END_IF
    END_FOR
    IF hits <> 1 THEN
        _M_RejectConfigSet(Scope := record.Scope, Key := record.WriteKey); RETURN;
    END_IF
END_FOR
// Station sets may carry a subset; a Model bank or Line calendar is complete.
IF (Info.Kind <> E_ConfigKind.STATION_CFG) AND (Info.RecordCount <> expectedInfo.RecordCount) THEN
    _M_RejectConfigSet(Scope := Info.RootIdentity, Key := Info.SetName); RETURN;
END_IF
_M_ValidateSetShape := TRUE;
END_METHOD

// Append an inactive provider record. Live recipe and existing ordinals stay fixed.
METHOD CreateModel : BOOL
VAR_INPUT
    ModelCode : STRING(160);
    SourceIndex : UDINT;
    FromSet : BOOL;
    SetName : STRING(80);
END_VAR
VAR
    i : INT;
    info : ST_ConfigSetInfo;
    record : ST_ConfigRecord;
    source : I_ConfigStore;
    sourceName : STRING(80);
END_VAR
CreateModel := FALSE;
IF NOT _M_ConfigRestored() THEN
    RETURN;
END_IF
_exportNext := 0;
_M_SyncModelCatalog();
IF (_modelCatalog = 0) OR (_pModelRegion = 0) OR (_modelRegionSize < SIZEOF(UINT))
OR (ModelCode = '') OR (LEN(ModelCode) > 64) OR (AvailableModelCount >= ModelCapacity)
OR NOT Access.PermitsLogged(Gate := E_GatedAction.CONFIG_SET) THEN RETURN; END_IF
FOR i := 1 TO AvailableModelCount DO
    IF AvailableModels[i].ModelCode = ModelCode THEN RETURN; END_IF
END_FOR
// The exact bytes being validated are copied into the existing view buffer.
IF NOT _M_CaptureConfig(SetName := '_validation', Kind := E_ConfigKind.PAR_CFG,
        ModelIndex := SourceIndex) THEN RETURN; END_IF
source := _snapshot;
sourceName := '_validation';
IF FromSet THEN
    IF _configStore = 0 THEN RETURN; END_IF
    IF NOT _M_CopySet(SetName := SetName) THEN RETURN; END_IF
    IF NOT _loadSnapshot.M_ReadInfo(SetName := SetName, Info := info) THEN RETURN; END_IF
    IF info.Kind <> E_ConfigKind.PAR_CFG THEN RETURN; END_IF
    IF NOT _M_ValidateSetShape(Store := _loadSnapshot, Info := info,
            AnyRevision := FALSE) THEN RETURN; END_IF
    source := _loadSnapshot;
    sourceName := SetName;
END_IF
IF NOT source.M_ReadInfo(SetName := sourceName, Info := info) THEN RETURN; END_IF
MEMCPY(destAddr := ADR(_modelBuf), srcAddr := _pModelRegion, n := _modelRegionSize);
IF SourceIndex > 0 THEN
    IF AvailableModels[SourceIndex].ModelCode <> Model.ModelCode THEN
    IF NOT _modelProvider.Load(ModelCode := AvailableModels[SourceIndex].ModelCode,
            RecipeKey := _modelKey, pParCfg := ADR(_modelBuf), Size := _modelRegionSize) THEN RETURN; END_IF
    END_IF
END_IF
_pModelView := ADR(_modelBuf);
FOR i := 1 TO info.RecordCount DO
    IF NOT source.M_ReadRecord(SetName := sourceName, Index := i, Record := record) THEN EXIT; END_IF
    // A provider with one root record cannot clone another owner's recipe bank.
    IF NOT _M_OwnsModelRecord(Record := record) THEN EXIT; END_IF
    IF NOT Access.M_PermitsLevelLogged(Required := _M_DataLevelOf(TargetPath := record.Scope,
            WriteKey := record.WriteKey, ForWrite := FALSE)) THEN EXIT; END_IF
    IF NOT Access.M_PermitsLevelLogged(Required := _M_DataLevelOf(TargetPath := record.Scope,
            WriteKey := record.WriteKey, ForWrite := TRUE)) THEN EXIT; END_IF
    IF NOT SUPER^.M_ApplyConfigWrite(Scope := record.Scope, WriteKey := record.WriteKey,
            Revision := record.Revision, TextValue := record.ValueText, RootReady := TRUE) THEN EXIT; END_IF
END_FOR
_pModelView := 0;
IF i <= info.RecordCount THEN RETURN; END_IF
CreateModel := _modelCatalog.M_CreateModel(ModelCode := ModelCode, RecipeKey := _modelKey,
    pData := ADR(_modelBuf), Size := _modelRegionSize);
IF CreateModel THEN
    _M_SyncModelCatalog();
    _M_MarkPersistPending();
END_IF
END_METHOD

METHOD ExportCurrentConfig : BOOL
VAR_INPUT
    SetName : STRING(80);
    Kind : E_ConfigKind;
    ModelIndex : UDINT;
    Token : STRING(160);
END_VAR
VAR
    info : ST_ConfigSetInfo;
    record : ST_ConfigRecord;
    i : INT;
END_VAR
ExportCurrentConfig := FALSE;
_exportNext := 0;
ConfigSetDocument := '';
ConfigSetDocumentLines := 0;
IF (Token = '') OR Access.ReqLogout
OR NOT Access.Permits(Gate := E_GatedAction.CONFIG_SET) THEN RETURN; END_IF
IF NOT _M_CaptureConfig(SetName := SetName, Kind := Kind, ModelIndex := ModelIndex) THEN RETURN; END_IF
_snapshot.M_ReadInfo(SetName := SetName, Info := info);
FOR i := 1 TO info.RecordCount DO
    _snapshot.M_ReadRecord(SetName := SetName, Index := i, Record := record);
    IF NOT Access.M_PermitsLevel(Required := _M_DataLevelOf(TargetPath := record.Scope,
            WriteKey := record.WriteKey, ForWrite := FALSE)) THEN RETURN; END_IF
END_FOR
_exportToken := Token;
_exportSession := Access.SessionGeneration;
_exportName := SetName;
_exportNext := 1;
ConfigSetDocument := _setJson.M_Header(Info := info);
ConfigSetDocumentLine := 0;
ConfigSetDocumentLines := info.RecordCount;
ExportCurrentConfig := ConfigSetDocument <> '';
END_METHOD

METHOD PRIVATE _M_ExportSnapshotLine : BOOL
VAR_INPUT
    SetName : STRING(80);
    Line : INT;
    Token : STRING(160);
END_VAR
VAR
    info : ST_ConfigSetInfo;
    record : ST_ConfigRecord;
END_VAR
_M_ExportSnapshotLine := FALSE;
ConfigSetDocument := '';
ConfigSetDocumentLines := 0;
IF (_exportNext = 0) OR (Line <> _exportNext) OR (Token <> _exportToken)
OR (_exportSession <> Access.SessionGeneration) OR (SetName <> _exportName)
OR Access.ReqLogout
OR NOT Access.Permits(Gate := E_GatedAction.CONFIG_SET) THEN
    _exportNext := 0; RETURN;
END_IF
IF NOT _snapshot.M_ReadInfo(SetName := SetName, Info := info)
OR NOT _snapshot.M_ReadRecord(SetName := SetName, Index := Line, Record := record) THEN
    _exportNext := 0; RETURN;
END_IF
IF NOT Access.M_PermitsLevel(Required := _M_DataLevelOf(TargetPath := record.Scope,
        WriteKey := record.WriteKey, ForWrite := FALSE)) THEN
    _exportNext := 0; RETURN;
END_IF
ConfigSetDocument := _setJson.M_Record(Record := record);
ConfigSetDocumentLine := Line;
ConfigSetDocumentLines := info.RecordCount;
_exportNext := _exportNext + 1;
IF Line = info.RecordCount THEN _exportNext := 0; END_IF
_M_ExportSnapshotLine := ConfigSetDocument <> '';
END_METHOD

END_FUNCTION_BLOCK

// ---- BaseClasses/FB_CompositeModuleBase.TcPOU
// Core §2.2 / §8.2 — CM lifecycle + child registry + first-out rollup.
// An EM type registers its children in Setup (_M_Register), ticks them every scan
// (_M_TickChildren, so status stays live whether or not a command runs — Annex B),
// and adopts the first faulted child's diagnostic verbatim (_M_RollupFault).
FUNCTION_BLOCK ABSTRACT FB_CompositeModuleBase EXTENDS FB_ModuleBase
VAR
    {attribute 'OPC.UA.DA' := '0'}
    _children : ARRAY[1..PL_Fraktal.MAX_EM_CHILDREN] OF I_Module;
    _nChild   : INT;
END_VAR

Cyclic();

// called from the type's Setup (Core §3.11); bounds-checked per Core §5.6
METHOD PROTECTED _M_Register : BOOL
VAR_INPUT
    Child : I_Module;
END_VAR
IF (Child = 0) OR (_nChild >= PL_Fraktal.MAX_EM_CHILDREN) THEN
    _M_Register := FALSE;
    RETURN;
END_IF
_nChild := _nChild + 1;
_children[_nChild] := Child;
_M_Register := TRUE;
END_METHOD

METHOD PrepareRecipe : BOOL
VAR_INPUT
    Model : ST_ModelId;
END_VAR
VAR
    i, j : INT;
END_VAR
PrepareRecipe := TRUE;
FOR i := 1 TO _nChild DO
    IF (_children[i] <> 0) AND_THEN NOT _children[i].PrepareRecipe(Model := Model) THEN
        PrepareRecipe := FALSE;
        FOR j := 1 TO i DO
            IF _children[j] <> 0 THEN _children[j].AbortRecipe(); END_IF
        END_FOR
        RETURN;
    END_IF
END_FOR
END_METHOD

METHOD CommitRecipe
VAR
    i : INT;
END_VAR
FOR i := 1 TO _nChild DO
    IF _children[i] <> 0 THEN _children[i].CommitRecipe(); END_IF
END_FOR
END_METHOD

METHOD AbortRecipe
VAR
    i : INT;
END_VAR
FOR i := 1 TO _nChild DO
    IF _children[i] <> 0 THEN _children[i].AbortRecipe(); END_IF
END_FOR
END_METHOD

// Core §8.2 — adopt the FIRST faulted child's first-out (reason + child SourcePath)
METHOD PROTECTED _M_RollupFault : BOOL
VAR
    i : INT;
END_VAR
_M_RollupFault := FALSE;
FOR i := 1 TO _nChild DO
    IF _children[i] <> 0 AND_THEN _children[i].FaultActive THEN
        _M_FaultDiag(_children[i].GetFaultSummary());
        _M_RollupFault := TRUE;
        RETURN;
    END_IF
END_FOR
END_METHOD

// Core §8.2/§6.1 HELD — the hold analogue of _M_RollupFault: adopt the FIRST held
// child's declared-wait reason (with the child's SourcePath) so this composite is
// held-and-explained rather than silently BUSY. No ERROR, no alarm: a hold rolls up
// as information, and clears itself when the child resumes.
METHOD PROTECTED _M_RollupHold : BOOL
VAR
    i : INT;
END_VAR
_M_RollupHold := FALSE;
FOR i := 1 TO _nChild DO
    IF _children[i] <> 0 AND_THEN _children[i].HoldActive THEN
        _M_HoldDiag(Diag := _children[i].GetFaultSummary());
        _M_RollupHold := TRUE;
        RETURN;
    END_IF
END_FOR
END_METHOD

// Core §6.1/§8.3(b) — releasing a composite's command releases the whole subtree:
// a frozen chain leaves commands asserted at every tier it had reached, and any one
// of them left high blocks that module's next command edge. Recursive by
// construction, so a nested EM needs no per-type recovery code.
METHOD M_ReleaseCommand : BOOL
M_ReleaseCommand := SUPER^.M_ReleaseCommand();
_M_ReleaseChildCommands();
END_METHOD

// Core §6.1/§8.3(b) — drop every registered child's command latch (recursively).
// Used by the recovery reset: the mode chain that issued those commands is no longer
// running, so nothing else will ever clear them (Core §6.8 chains hold the child's
// Execute in the step that issued it).
METHOD PROTECTED _M_ReleaseChildCommands
VAR
    i : INT;
END_VAR
FOR i := 1 TO _nChild DO
    IF _children[i] <> 0 THEN
        _children[i].M_ReleaseCommand();
    END_IF
END_FOR
END_METHOD

// children always tick so their status stays live (Annex B §B.3)
METHOD PROTECTED _M_TickChildren
VAR
    i : INT;
END_VAR
FOR i := 1 TO _nChild DO
    IF _children[i] <> 0 THEN
        _children[i].Cyclic();
    END_IF
END_FOR
END_METHOD

PROPERTY ModuleType : E_ModuleType
GET
ModuleType := E_ModuleType.NONE;
END_GET
END_PROPERTY

// §3.10.2 — own facets first, then every registered child, depth-first in
// registration order so the manifest walk is deterministic across requests.
METHOD M_AppendConfig : BOOL
VAR_INPUT
    Pager : REFERENCE TO FB_ConfigPager;
END_VAR
VAR
    i    : INT;
    iCfg : I_ConfigSource;
END_VAR
M_AppendConfig := SUPER^.M_AppendConfig(Pager := Pager);
FOR i := 1 TO _nChild DO
    IF _children[i] <> 0 THEN
        IF __QUERYINTERFACE(_children[i], iCfg) THEN
            iCfg.M_AppendConfig(Pager := Pager);
        END_IF
    END_IF
END_FOR
END_METHOD

// §3.8b — own registrations first, then every registered child, in the same
// depth-first order as M_AppendConfig. Scope makes the walk unambiguous: at most
// one module answers, and the first TRUE ends it.
METHOD M_ApplyConfigWrite : BOOL
VAR_INPUT
    Scope     : STRING(255);
    WriteKey  : STRING(160);
    Revision  : UDINT;
    TextValue : STRING(255);
    RootReady : BOOL;
END_VAR
VAR
    i    : INT;
    iCfg : I_ConfigSource;
END_VAR
M_ApplyConfigWrite := SUPER^.M_ApplyConfigWrite(Scope := Scope,
    WriteKey := WriteKey, Revision := Revision, TextValue := TextValue,
    RootReady := RootReady);
IF M_ApplyConfigWrite THEN
    RETURN;
END_IF
FOR i := 1 TO _nChild DO
    IF _children[i] <> 0 THEN
        IF __QUERYINTERFACE(_children[i], iCfg) THEN
            IF iCfg.M_ApplyConfigWrite(Scope := Scope, WriteKey := WriteKey,
                    Revision := Revision, TextValue := TextValue,
                    RootReady := RootReady) THEN
                M_ApplyConfigWrite := TRUE;
                RETURN;
            END_IF
        END_IF
    END_IF
END_FOR
END_METHOD

// §3.8d - the access walk is the write walk: same order, same "first owner
// answers TRUE" rule, so the level checked is the level of the value written.
METHOD M_ConfigAccessOf : BOOL
VAR_INPUT
    Scope    : STRING(255);
    WriteKey : STRING(160);
END_VAR
VAR_IN_OUT
    Grant : ST_ConfigAccess;
END_VAR
VAR
    i    : INT;
    iCfg : I_ConfigSource;
END_VAR
M_ConfigAccessOf := SUPER^.M_ConfigAccessOf(Scope := Scope, WriteKey := WriteKey,
    Grant := Grant);
IF M_ConfigAccessOf THEN
    RETURN;
END_IF
FOR i := 1 TO _nChild DO
    IF _children[i] <> 0 THEN
        IF __QUERYINTERFACE(_children[i], iCfg) THEN
            IF iCfg.M_ConfigAccessOf(Scope := Scope, WriteKey := WriteKey,
                    Grant := Grant) THEN
                M_ConfigAccessOf := TRUE;
                RETURN;
            END_IF
        END_IF
    END_IF
END_FOR
END_METHOD

// §3.8c - the capture walk is the write walk. Same order, same "first owner
// answers TRUE" rule, so a capture reaches exactly the module a write would.
METHOD M_ApplyCapture : BOOL
VAR_INPUT
    Scope     : STRING(255);
    WriteKey  : STRING(160);
    Revision  : UDINT;
    RootReady : BOOL;
END_VAR
VAR
    i    : INT;
    iCfg : I_ConfigSource;
END_VAR
M_ApplyCapture := SUPER^.M_ApplyCapture(Scope := Scope, WriteKey := WriteKey,
    Revision := Revision, RootReady := RootReady);
IF M_ApplyCapture THEN
    RETURN;
END_IF
FOR i := 1 TO _nChild DO
    IF _children[i] <> 0 THEN
        IF __QUERYINTERFACE(_children[i], iCfg) THEN
            IF iCfg.M_ApplyCapture(Scope := Scope, WriteKey := WriteKey,
                    Revision := Revision, RootReady := RootReady) THEN
                M_ApplyCapture := TRUE;
                RETURN;
            END_IF
        END_IF
    END_IF
END_FOR
END_METHOD

// §3.8b — the staging walk is the write walk. Same order, same "first owner
// answers TRUE" rule, so a record that stages here is the record that will
// apply there, on the same module.
METHOD M_StageConfigWrite : BOOL
VAR_INPUT
    Scope     : STRING(255);
    WriteKey  : STRING(160);
    Revision  : UDINT;
    TextValue : STRING(255);
    RootReady : BOOL;
END_VAR
VAR
    i    : INT;
    iCfg : I_ConfigSource;
END_VAR
M_StageConfigWrite := SUPER^.M_StageConfigWrite(Scope := Scope,
    WriteKey := WriteKey, Revision := Revision, TextValue := TextValue,
    RootReady := RootReady);
IF M_StageConfigWrite THEN
    RETURN;
END_IF
FOR i := 1 TO _nChild DO
    IF _children[i] <> 0 THEN
        IF __QUERYINTERFACE(_children[i], iCfg) THEN
            IF iCfg.M_StageConfigWrite(Scope := Scope, WriteKey := WriteKey,
                    Revision := Revision, TextValue := TextValue,
                    RootReady := RootReady) THEN
                M_StageConfigWrite := TRUE;
                RETURN;
            END_IF
        END_IF
    END_IF
END_FOR
END_METHOD

// §3.8b — own loss first, then the children in registration order. One loss per
// call: the root drains until FALSE, so a subtree that lost several images
// annunciates each of them with its own owning path rather than one summary
// that names nobody.
METHOD M_TakeRestoreLoss : BOOL
VAR_OUTPUT
    Path     : STRING(80);
    Expected : UINT;
    Found    : UINT;
END_VAR
VAR
    i    : INT;
    iCfg : I_ConfigSource;
END_VAR
M_TakeRestoreLoss := SUPER^.M_TakeRestoreLoss(Path => Path,
    Expected => Expected, Found => Found);
IF M_TakeRestoreLoss THEN
    RETURN;
END_IF
FOR i := 1 TO _nChild DO
    IF _children[i] <> 0 THEN
        IF __QUERYINTERFACE(_children[i], iCfg) THEN
            IF iCfg.M_TakeRestoreLoss(Path => Path, Expected => Expected,
                    Found => Found) THEN
                M_TakeRestoreLoss := TRUE;
                RETURN;
            END_IF
        END_IF
    END_IF
END_FOR
END_METHOD

// §7.6.1 - own registration first, then every registered child in the same
// depth-first order as the config walk. Scope makes it unambiguous: at most one
// module answers and the first TRUE ends it.
METHOD M_ApplyManual : BOOL
VAR_INPUT
    Scope : STRING(255);
    Value : DINT;
END_VAR
VAR
    i    : INT;
    iMan : I_ManualTarget;
END_VAR
M_ApplyManual := SUPER^.M_ApplyManual(Scope := Scope, Value := Value);
IF M_ApplyManual THEN
    RETURN;
END_IF
FOR i := 1 TO _nChild DO
    IF _children[i] <> 0 THEN
        IF __QUERYINTERFACE(_children[i], iMan) THEN
            IF iMan.M_ApplyManual(Scope := Scope, Value := Value) THEN
                M_ApplyManual := TRUE;
                RETURN;
            END_IF
        END_IF
    END_IF
END_FOR
END_METHOD

// §7.6.1a - the held walk is the manual walk. Same order, same "first owner
// answers TRUE" rule, so a hold reaches exactly the module a one-shot would.
METHOD M_ApplyHeld : BOOL
VAR_INPUT
    Scope  : STRING(255);
    Value  : DINT;
    Enable : ST_ManualEnableStatus;
END_VAR
VAR
    i    : INT;
    iMan : I_ManualTarget;
END_VAR
M_ApplyHeld := SUPER^.M_ApplyHeld(Scope := Scope, Value := Value,
    Enable := Enable);
IF M_ApplyHeld THEN
    RETURN;
END_IF
FOR i := 1 TO _nChild DO
    IF _children[i] <> 0 THEN
        IF __QUERYINTERFACE(_children[i], iMan) THEN
            IF iMan.M_ApplyHeld(Scope := Scope, Value := Value,
                    Enable := Enable) THEN
                M_ApplyHeld := TRUE;
                RETURN;
            END_IF
        END_IF
    END_IF
END_FOR
END_METHOD

END_FUNCTION_BLOCK

// ---- BaseClasses/FB_ModuleBase.TcPOU
// Core §2.2 / §6.1 — the PLCopen lifecycle written ONCE (template method).
// A concrete type EXTENDS this base, declares its Command/HAL/ParCfg members, and
// overrides only _M_Dispatch (+ optionally hooks and recipe transaction methods).
// Edge handling, ExecState mapping, Execute-drop reset, ErrorID publication, and
// abort routing are inherited. Conformance rows T1/T4 (Core §5.7) are satisfied here
// and proven once in FB_Base_Tests.
FUNCTION_BLOCK ABSTRACT FB_ModuleBase IMPLEMENTS I_Module, I_ConfigSource, I_ManualTarget
VAR_INPUT
    Execute : BOOL;    // rising edge starts the command (Core §6.1)
    Abort   : BOOL;    // requests a controlled abort
END_VAR
VAR_OUTPUT
    Busy    : BOOL;
    Done    : BOOL;
    Error   : BOOL;
    Aborted : BOOL;
    // Core §6.1 — ISA-88 HELD, orthogonal to the terminal states: BUSY, outputs
    // withdrawn, deliberately not progressing while a declared condition is
    // unsatisfied. Deliberately NOT an E_ExecState ordinal: that enum is transport
    // contract (§3.10(a')) and the HMI mirrors its ordinals, so HELD is published
    // as its own flag beside Busy/Done/Error/Aborted and never renumbers the set.
    Held    : BOOL;
    // §3.13 — does this module publish a sequence flow chart? A type that has
    // no meaningful chain leaves it FALSE and the HMI omits the tab entirely;
    // FB_UnitBase defaults it TRUE and a Unit may vary it per mode.
    SequenceViewEnabled : BOOL;
    ErrorID : DWORD;   // = TO_DWORD(first-out ReasonCode), Core §8.8
    // §3.12 — derived state published by this module: facts recomputed from the
    // real state underneath, every scan. Distinct from OutCmd, which is what a
    // command produced and stays latched until the next one.
    StateFlags : ARRAY[1..PL_Fraktal.MAX_STATE_FLAGS] OF ST_StateFlag;
    StateFlagCount : INT;              // highest index published (§8.4 bounded)
END_VAR
VAR_OUTPUT
    Status : ST_ModuleStatus;   // Core §3.10(a')/§6.9(a) — the OPC UA data mirror
    Timing : ST_ModuleTiming;   // Core §8.11.4(a) — per-command timing, captured here once
    // §3.10.2 — static facets stay OFF the cyclic OPC UA tree and are served
    // through the QUERY_CONFIG manifest instead (M_AppendConfig).
    {attribute 'OPC.UA.DA' := '0'}
    Nameplate   : ST_Nameplate;  // §3.10.1 asset identity (set at Setup; empty = none)
    {attribute 'OPC.UA.DA' := '0'}
    Catalog     : ARRAY[1..PL_Fraktal.MAX_CMD_CATALOG] OF ST_CommandInfo;  // §7.6.1 published command list
    {attribute 'OPC.UA.DA' := '0'}
    CatalogCount: INT;
    Safety       : ST_SafetyStatus;       // §9 optional read-only safety facet (Present=FALSE if absent)
    ControlPower : ST_ControlPowerStatus; // §9 optional control/power facet
END_VAR
VAR
    _name  : STRING(80);
    _exec  : E_ExecState := E_ExecState.READY;
    _step  : INT;
    _diag  : ST_Diagnostic;
    _rTrig : R_TRIG;
    _abortErrTrig : R_TRIG;
    _initialized : BOOL;
    _prevExec   : E_ExecState;
    _manualCmd  : DINT;          // §7.6.1 pending manual command value (0 = none)
    _manualReq  : BOOL;
    _manualActive : BOOL;        // one-shot manual request owns Execute until terminal state
    _cmdArmed   : BOOL;          // terminal state came from a command; gates the §6.1 reset
    _stateTouched : ARRAY[1..PL_Fraktal.MAX_STATE_FLAGS] OF BOOL;   // §3.12 published this scan
    _cmdId      : DINT;          // set by _M_TagCommand (one line per type, §8.11.4(a))
    _cmdLabel   : STRING(120);
    _tCmdStart  : DWORD;         // monotonic ms at command start (TC3 §8.11)
    _holdReq    : BOOL;          // §6.1 HELD: re-asserted by dispatch every scan it holds
    _holdSince  : DATE_AND_TIME; // hold onset, preserved across scans (§8.8 Since)
    _holdTimeSynchronized : BOOL;
    // §3.8b/§3.10.2 — the editable values this module has registered about
    // itself. One record serves both directions: the manifest publishes the
    // capability from it and a write applies through it, so the metadata a
    // client validated against and the target actually written cannot drift
    // apart (§1.1 O1). Off the cyclic tree — pTarget must never reach a client.
    {attribute 'OPC.UA.DA' := '0'}
    _configWrite  : ARRAY[1..PL_Fraktal.MAX_CONFIG_WRITES] OF ST_ConfigWriteDef;
    {attribute 'OPC.UA.DA' := '0'}
    _nConfigWrite : INT;
    {attribute 'OPC.UA.DA' := '0'}
    _pConfigWrite : POINTER TO ST_ConfigWriteDef;
    _configCapacity : INT := PL_Fraktal.MAX_CONFIG_WRITES;
    // §3.8a - this module's own recipe record, and the record a request is
    // viewing instead of it (0 = the live one). See _M_SetModelRegion.
    {attribute 'OPC.UA.DA' := '0'}
    _pModelRegion : PVOID;
    _modelRegionSize : UDINT;
    {attribute 'OPC.UA.DA' := '0'}
    _pModelView : PVOID;
    // §3.8b — one restore-loss slot. ONE, not a list: a module with two retained
    // structures that both lost their schema lost them for the same reason (its
    // own layout changed), and one annunciation naming the module is exactly
    // what the operator needs. The slot is cleared as the root takes it, so the
    // event is raised exactly once per boot.
    {attribute 'OPC.UA.DA' := '0'}
    _restoreLost     : BOOL;
    {attribute 'OPC.UA.DA' := '0'}
    _restoreExpected : UINT;
    {attribute 'OPC.UA.DA' := '0'}
    _restoreFound    : UINT;
END_VAR

// FB body just runs the lifecycle; parents may call the instance or Cyclic() (I_Module)
Cyclic();

// Core §6.1 — edge -> hooks -> dispatch -> map -> Execute-drop reset
METHOD Cyclic : BOOL
VAR
    commandStarted : BOOL;
END_VAR
commandStarted := FALSE;
// Execute-drop reset (Core §6.1): a COMMAND-produced terminal state published in
// an earlier scan plus Execute low resets to READY BEFORE this scan's mapping, so
// the outputs go idle in the same call. A completion later this scan still maps
// its one-cycle DONE/ERROR/ABORTED pulse first (PLCopen). Faults raised OUTSIDE a
// command (recipe/config at Setup, cyclic condition monitors) latch (§3.8/§8.3):
// Execute was never high, so the handshake reset does not consume them.
IF (NOT Execute) AND _cmdArmed
AND ((_exec = E_ExecState.DONE) OR (_exec = E_ExecState.ERROR) OR (_exec = E_ExecState.ABORTED)) THEN
    _exec := E_ExecState.READY;
    _cmdArmed := FALSE;
END_IF

_rTrig(CLK := Execute);
// A fresh command edge may also RETRY from a latched non-command fault: the edge
// clears the diagnostic and re-runs validation, which re-faults if the cause remains.
IF _rTrig.Q AND ((_exec = E_ExecState.READY)
    OR ((_exec = E_ExecState.ERROR) AND NOT _cmdArmed)) THEN
    _exec := E_ExecState.BUSY;      // ParCmd of the concrete type is latched on this edge
    _cmdArmed := TRUE;
    _step := 10;
    _M_ClearDiag();
    _tCmdStart := TIME_TO_DWORD(TIME());          // §8.11.4(a) command-timing start
    commandStarted := TRUE;
END_IF

IF NOT _initialized THEN
    _initialized := TRUE;
    OnInit();                        // Core §3.14 one-shot for every module tier
END_IF
IF commandStarted THEN
    OnCommandStart();                // one-shot after init, before cyclic/dispatch
END_IF
_M_SweepStateFlags();                // §3.12 last scan's flags resolve here
OnCyclic();                          // Core §3.14 hook: background management, no outputs

IF Abort AND (_exec = E_ExecState.BUSY) THEN
    OnAbort();                       // Core §3.14 hook: device-safe abort action
END_IF
_abortErrTrig(CLK := Abort AND (_exec = E_ExecState.ERROR));
IF _abortErrTrig.Q THEN
    OnAbortInError();                // distinct recovery hook; ERROR remains latched
END_IF

IF _exec = E_ExecState.BUSY THEN
    _M_Dispatch();                   // the ONLY thing a type must write (Core §2.2)
END_IF

// §6.1 HELD resolution — level-based, exactly like an interlock: a hold lasts only
// while this scan's dispatch re-asserted it, so a restored condition resumes by
// itself with no per-type "clear the hold" code to forget. A hold never survives
// leaving BUSY, and a fault raised in the same scan keeps its own diagnostic.
IF Held AND (NOT _holdReq) AND (_exec = E_ExecState.BUSY) THEN
    _M_ClearDiag();                  // the declared condition returned
END_IF
Held := _holdReq AND (_exec = E_ExecState.BUSY);
_holdReq := FALSE;

// §8.11.4(a) — close the command's timing row on leaving BUSY (DONE/ERROR/ABORTED)
IF (_prevExec = E_ExecState.BUSY) AND (_exec <> E_ExecState.BUSY) THEN
    _M_RecordCmdTiming(TIME_TO_DWORD(TIME()) - _tCmdStart);   // wrap-safe diff (TC3 §8.11)
END_IF
_prevExec := _exec;

Busy    := (_exec = E_ExecState.BUSY);
Done    := (_exec = E_ExecState.DONE);
Error   := (_exec = E_ExecState.ERROR);
Aborted := (_exec = E_ExecState.ABORTED);
ErrorID := TO_DWORD(_diag.ReasonCode);

// §6.9(a)/§3.10(a') — refresh the data mirror: properties are invisible to the
// OPC UA namespace, so everything the HMI binds is published here as DATA
Status.ModuleType  := ModuleType;
Status.State       := _exec;
Status.FaultActive := (_exec = E_ExecState.ERROR);
Status.Diagnostic  := _diag;
_M_PublishStatus();              // tier-specific overlay after the common mirror is final

// A manual command is a one-shot use of the same PLCopen lifecycle. Keep the
// terminal state visible for this scan, then drop Execute for next-scan reset.
IF _manualActive AND ((_exec = E_ExecState.DONE) OR (_exec = E_ExecState.ERROR) OR (_exec = E_ExecState.ABORTED)) THEN
    Execute := FALSE;
    _manualActive := FALSE;
END_IF
Cyclic := TRUE;
END_METHOD

// Core §8.2/§6.9 — this node's first-out (composites override via rollup in the EM base)
METHOD GetFaultSummary : ST_Diagnostic
GetFaultSummary := _diag;
END_METHOD

// Core §3.14 hook — optional override: device-safe abort action.
// Override contract (Core §3.14.2): call SUPER^.OnAbort() FIRST and keep its return.
METHOD PROTECTED OnAbort : DINT
_exec := E_ExecState.ABORTED;
_step := 0;
OnAbort := 0;
END_METHOD

// Core §3.14 — optional error-state abort/recovery action. ERROR remains latched
// until Execute drops. Overrides call SUPER^.OnAbortInError() first.
METHOD PROTECTED OnAbortInError : DINT
OnAbortInError := 0;
END_METHOD

// Core §3.14 — first operational scan, after Setup/recipe load.
// Overrides call SUPER^.OnInit() first and propagate its return.
METHOD PROTECTED OnInit : DINT
OnInit := 0;
END_METHOD

// Core §3.14 hook — optional override: per-scan background management (idempotent,
// no direct outputs). Override contract: call SUPER^.OnCyclic() FIRST, keep return.
METHOD PROTECTED OnCyclic : DINT
OnCyclic := 0;
END_METHOD

// Core §3.14 hook — one-shot on each accepted Execute rising edge, after OnInit
// and before OnCyclic/_M_Dispatch. Overrides call SUPER^.OnCommandStart() first.
// Use for command-local wiring/reset only; process behavior belongs in dispatch.
METHOD PROTECTED OnCommandStart : DINT
OnCommandStart := 0;
END_METHOD

// Core §3.8 — types with ParCfg load into staging here.
METHOD PrepareRecipe : BOOL
VAR_INPUT
    Model : ST_ModelId;
END_VAR
PrepareRecipe := TRUE;
END_METHOD

METHOD CommitRecipe
END_METHOD

METHOD AbortRecipe
END_METHOD

// Core §3.2 — generic DINT command path; the catalog is the supported set.
// Concrete dispatch consumes the inherited manual request, so typed/generic/HMI
// paths share validation, timing, interlocks, and the PLCopen lifecycle.
METHOD ExecuteCommand : BOOL
VAR_INPUT
    Command : DINT;
END_VAR
ExecuteCommand := ManualCommand(Value := Command);
END_METHOD

// Core §3.2/§6.1 — method form of the inherited abort route.
METHOD AbortCommand : BOOL
AbortCommand := FALSE;
IF _exec <> E_ExecState.BUSY THEN
    RETURN;
END_IF
OnAbort();
_exec := E_ExecState.ABORTED;
_step := 0;
AbortCommand := TRUE;
END_METHOD

METHOD PROTECTED _M_ClearDiag
_diag.ReasonCode  := E_Reason.NONE;
_diag.Description := '';
_diag.IoTag := '';
_diag.IoAddress := '';
_diag.TimeSynchronized := FALSE;
END_METHOD

// Core §6.1 — successful completion (the concrete type publishes OutCmd before calling)
METHOD PROTECTED _M_Complete
_exec := E_ExecState.DONE;
_step := 0;
_M_ClearDiag();
END_METHOD

// Core §2.2 — THE extension point: the type's CASE _step device logic,
// calling _M_Fault / _M_FaultDiag / _M_Complete.
METHOD PROTECTED ABSTRACT _M_Dispatch
END_METHOD

// Core §6.9 — stamp the first-out reason and hold in ERROR
METHOD PROTECTED _M_Fault
VAR_INPUT
    Reason : E_Reason;
    Text   : STRING(255);
END_VAR
_diag.ReasonCode  := Reason;
_diag.Description := Text;
_diag.SourcePath  := _name;
_diag.IoTag       := '';
_diag.IoAddress   := '';
_diag.Severity    := E_Severity.MED;
_diag.Category    := E_Category.PROCESS;
F_RationalizeDiagnostic(Diag := _diag);
_diag.Since       := F_Now();       // synchronized clock (Core §2.7)
_diag.TimeSynchronized := F_TimeSynchronized();
_exec := E_ExecState.ERROR;
_step := 0;
END_METHOD

// Core §8.2 — adopt a ready-made diagnostic verbatim (rollup / connector reason)
METHOD PROTECTED _M_FaultDiag
VAR_INPUT
    Diag : ST_Diagnostic;
END_VAR
_diag := Diag;
F_RationalizeDiagnostic(Diag := _diag);
_exec := E_ExecState.ERROR;
_step := 0;
END_METHOD

// called from the concrete type's Setup (Core §3.11); Name = browse path (Core §4.8)
METHOD PROTECTED _M_SetName
VAR_INPUT
    Name : STRING(80);
END_VAR
_name := Name;
Status.Name := Name;   // mirror (§3.10(a'))
END_METHOD

// Core §8.11.4(a) — fold the finished command into its timing row (find-or-allocate)
METHOD PRIVATE _M_RecordCmdTiming
VAR_INPUT
    DurMs : DWORD;
END_VAR
VAR
    i, slot : INT;
END_VAR
Timing.LastCmdTime := DWORD_TO_TIME(DurMs);
slot := 0;
FOR i := 1 TO PL_Fraktal.MAX_CMD_STATS DO
    IF (Timing.Rows[i].Count > 0) AND (Timing.Rows[i].Id = _cmdId) THEN
        slot := i;
        EXIT;
    ELSIF (slot = 0) AND (Timing.Rows[i].Count = 0) THEN
        slot := i;
    END_IF
END_FOR
IF slot = 0 THEN
    Timing.Truncated := TRUE;        // fixed array, never grown at runtime (§8.11.4(e))
ELSE
    Timing.Rows[slot].Id    := _cmdId;
    Timing.Rows[slot].Label := _cmdLabel;
    F_TimingUpdate(Row := Timing.Rows[slot], DurMs := DurMs);
END_IF
END_METHOD

// §3.12 — publish a DERIVED state flag and return it, so the assignment reads
// exactly as it would without the framework:
//
//     OutImm.Homed := _M_State(Idx := 1, Key := 'project.state.atHome',
//         Ok := Ram.OutImm.Retracted AND Door.OutImm.Retracted);
//
// What the call adds over a bare assignment is everything the operator and the
// HMI need and nobody wants to write per flag (§1.1 O1): the flag carries its
// own name, and the moment it last changed (§2.7), and it is published on a
// bounded generic table the HMI renders without knowing the module type (§3.13).
// Same shape as the §6.9(b) named condition wait, deliberately - one idiom for
// "a named boolean the framework publishes" (§1.1 O9).
//
// CALL IT UNCONDITIONALLY, every scan. A flag that stops being published goes
// Stale and its Value is forced FALSE on the next scan: state that nobody is
// computing is not a claim. That is the point of the mechanism - a latch left
// standing is exactly the failure it exists to prevent.
//
// Out-of-range Idx is skipped rather than faulted, matching _M_Await (§6.9(b)):
// the value still returns, so a mis-indexed flag loses its publication, never
// the machine logic that reads it.
METHOD PROTECTED _M_State : BOOL
VAR_INPUT
    Idx : INT;
    Key : STRING(120);
    Ok  : BOOL;
END_VAR
_M_State := Ok;
IF (Idx < 1) OR (Idx > PL_Fraktal.MAX_STATE_FLAGS) THEN
    RETURN;
END_IF
IF Idx > StateFlagCount THEN
    StateFlagCount := Idx;
END_IF
IF (StateFlags[Idx].Value <> Ok) OR (StateFlags[Idx].Key <> Key)
OR StateFlags[Idx].Stale THEN
    StateFlags[Idx].Since := F_Now();      // §2.7 synchronized clock
END_IF
StateFlags[Idx].Key   := Key;
StateFlags[Idx].Value := Ok;
StateFlags[Idx].Stale := FALSE;
_stateTouched[Idx] := TRUE;
END_METHOD

// §3.12 — resolve the previous scan's publications, before this scan re-publishes.
// A flag the owner stopped computing stops claiming; nothing has to be
// deregistered when a module stops publishing one (§1.1 O1).
METHOD PRIVATE _M_SweepStateFlags
VAR
    i : INT;
END_VAR
FOR i := 1 TO StateFlagCount DO
    IF NOT _stateTouched[i] THEN
        StateFlags[i].Value := FALSE;
        StateFlags[i].Stale := TRUE;
    END_IF
    _stateTouched[i] := FALSE;
END_FOR
END_METHOD

// Core §8.11.4(a) — the ONE line a type adds for a per-command breakdown:
//   _M_TagCommand(TO_DINT(Command), '<label>');   (idempotent; scaffold includes it)
METHOD PROTECTED _M_TagCommand
VAR_INPUT
    Id    : DINT;
    Label : STRING(120);
END_VAR
_cmdId    := Id;
    _cmdLabel := Label;
END_METHOD

// Optional localizable HMI metadata; keys only, never operator prose.
METHOD PROTECTED _M_SetPresentation
VAR_INPUT
    DisplayNameKey : STRING(160);
    DescriptionKey : STRING(160);
    TypeKey : STRING(160);        // §7.1: the TYPE's key, never an instance variable
END_VAR
Status.DisplayNameKey := DisplayNameKey;
Status.DescriptionKey := DescriptionKey;
Status.TypeKey := TypeKey;
END_METHOD

// Core §8.8 band-extensibility: fault with a per-type band code (DINT constant).
// E_Reason is deliberately non-strict, so the numeric assignment is contract, not a cast trick.
METHOD PROTECTED _M_FaultN
VAR_INPUT
    Code : DINT;          // registered band code (Core §8.8 registry)
    Text : STRING(255);
END_VAR
_diag.ReasonCode  := Code;    // non-strict enum accepts the band value (Core §8.8)
_diag.Description := Text;
_diag.SourcePath  := _name;
_diag.IoTag       := '';
_diag.IoAddress   := '';
_diag.Severity    := E_Severity.MED;
_diag.Category    := E_Category.PROCESS;
F_RationalizeDiagnostic(Diag := _diag);
_diag.Since       := F_Now();
_diag.TimeSynchronized := F_TimeSynchronized();
_exec := E_ExecState.ERROR;
_step := 0;
END_METHOD

// Type-band fault with the implicated schematic tag and terminal location.
METHOD PROTECTED _M_FaultIoN
VAR_INPUT
    Code : DINT;
    Text : STRING(255);
    IoTag : STRING(80);
    IoAddress : STRING(80);
END_VAR
_M_FaultN(Code := Code, Text := Text);
_diag.IoTag := IoTag;
_diag.IoAddress := IoAddress;
END_METHOD

// Core §6.1 HELD — suspend progress on a NAMED condition instead of faulting.
// Use it where the condition is expected operator or process behaviour rather than
// a defect: an interlock lost mid-motion, a hold-to-run permissive released. The
// module stays BUSY, so the owner keeps awaiting it and resumes when the condition
// returns; no ERROR, no MANUAL_RESET alarm, nothing to reset. Call it from dispatch
// EVERY scan the condition is unsatisfied — the base clears the hold as soon as a
// scan stops re-asserting it. Withdrawing the outputs stays the caller's job: only
// the device type knows which of its outputs are unsafe to leave energized.
METHOD PROTECTED _M_Hold
VAR_INPUT
    Reason : E_Reason;
    Text   : STRING(255);
END_VAR
IF NOT Held THEN
    _holdSince := F_Now();           // onset stamped once (§2.7 synchronized clock)
    _holdTimeSynchronized := F_TimeSynchronized();
END_IF
_diag.ReasonCode  := Reason;
_diag.Description := Text;
_diag.SourcePath  := _name;
_diag.IoTag       := '';
_diag.IoAddress   := '';
_diag.Severity    := E_Severity.LOW;   // a declared wait informs; it is not a fault (§8.1)
_diag.Category    := E_Category.PROCESS;
_diag.Since       := _holdSince;
_diag.TimeSynchronized := _holdTimeSynchronized;
_holdReq := TRUE;
END_METHOD

// Core §6.1 HELD / §8.2 — hold on a ready-made diagnostic (an interlock's first-out,
// or a held child's reason adopted by its parent). Keeps the originating SourcePath
// so the operator sees WHICH module is waiting on WHICH condition (§6.9).
METHOD PROTECTED _M_HoldDiag
VAR_INPUT
    Diag : ST_Diagnostic;
END_VAR
IF NOT Held THEN
    _holdSince := Diag.Since;        // the condition's own onset, not this scan
    _holdTimeSynchronized := Diag.TimeSynchronized;
END_IF
_diag := Diag;
_diag.Severity := E_Severity.LOW;
_diag.Since    := _holdSince;
_diag.TimeSynchronized := _holdTimeSynchronized;
_holdReq := TRUE;
END_METHOD

// Core §6.1/§8.3(b) — release a command this module can no longer be driven to
// finish, so the inherited Execute-drop reset clears a latched terminal state on
// the next scan. Deliberately does NOT touch _exec: that transition stays owned by
// Cyclic, preserving the §6.1 reset-provenance rule (IMPLEMENTATION_NOTES §47).
// A live cause therefore re-faults on the next command edge rather than vanishing.
METHOD M_ReleaseCommand : BOOL
// A command still BUSY (mid-motion, or HELD on a condition) needs cancelling, not
// just un-asserting: BUSY is not a terminal state, so the Execute-drop reset skips
// it and the §6.1 acceptance test (`_rTrig.Q AND _exec = READY`) would ignore every
// later command edge — the module would sit BUSY forever and the recovery sequence
// would wait on it. AbortCommand routes through OnAbort, so the device gets its own
// safe-stop action before the handshake unwinds.
IF _exec = E_ExecState.BUSY THEN
    AbortCommand();                  // -> ABORTED, then READY once Execute is low
END_IF
Execute := FALSE;
_manualReq    := FALSE;              // an unconsumed manual request must not fire later
_manualActive := FALSE;
M_ReleaseCommand := TRUE;
END_METHOD

PROPERTY HoldActive : BOOL
GET
HoldActive := Held;
END_GET
END_PROPERTY

PROPERTY FaultActive : BOOL
GET
FaultActive := (_exec = E_ExecState.ERROR);
END_GET
END_PROPERTY

PROPERTY ModuleType : E_ModuleType
GET
ModuleType := E_ModuleType.NONE;
END_GET
END_PROPERTY

PROPERTY Name : STRING(80)
GET
Name := _name;
END_GET
END_PROPERTY

PROPERTY State : E_ExecState
GET
State := _exec;
END_GET
END_PROPERTY

// §7.6.1 — register one manual command in the catalog (call in the module's init).
// Idempotent by Value: re-publishing a Value updates its label.
METHOD PROTECTED _M_PublishCommand
VAR_INPUT
    Value : DINT;
    Label : STRING(120);
END_VAR
VAR
    i : INT;
END_VAR
FOR i := 1 TO CatalogCount DO
    IF Catalog[i].Value = Value THEN
        Catalog[i].Label := Label;
        RETURN;
    END_IF
END_FOR
IF CatalogCount >= PL_Fraktal.MAX_CMD_CATALOG THEN
    RETURN;
END_IF
CatalogCount := CatalogCount + 1;
Catalog[CatalogCount].Value := Value;
Catalog[CatalogCount].Label := Label;
END_METHOD

// §7.6.1 - register a HELD manual command (a jog). Same catalog, same
// idempotence; the style tells the HMI to render press-and-hold and to route it
// to RequestHeldCommand instead of ExecuteCommand.
METHOD PROTECTED _M_PublishHeldCommand
VAR_INPUT
    Value : DINT;
    Label : STRING(120);
END_VAR
VAR
    i : INT;
END_VAR
_M_PublishCommand(Value := Value, Label := Label);
FOR i := 1 TO CatalogCount DO
    IF Catalog[i].Value = Value THEN
        Catalog[i].Style := E_CommandStyle.HELD;
        RETURN;
    END_IF
END_FOR
END_METHOD

// §7.6.1 - the entry point for a HELD manual command, called EVERY SCAN while
// the operator holds the control. Silence is a stop: a module that implements
// this shall stop the action when the calls stop, whether the operator let go or
// the transport died (O10 - a lost connection queues nothing).
//
// Enable carries the §9 manual-enable fact for actions that need one (motion
// with the guards open). It is STATUS, never authority: the module still applies
// its own interlocks, and the safety system remains what actually permits the
// movement. Modules with no held commands inherit this refusal unchanged.
METHOD RequestHeldCommand : BOOL
VAR_INPUT
    Value  : DINT;
    Enable : ST_ManualEnableStatus;
END_VAR
RequestHeldCommand := FALSE;   // no held commands on this type (§5.6 defined ELSE)
END_METHOD

// §7.6.1 — apply a manual command, routed THROUGH the normal command surface so
// interlocks/first-out/timing still apply (§3.2). The owning Unit is the single
// gate: it calls this ONLY after verifying MANUAL mode (§3.4) + MANUAL access
// (§7.7) and logs the §8.3 event. §7.6 Release<Function> is enforced by the
// module's own _M_Dispatch. Concrete modules read _manualReq/_manualCmd there.
METHOD ManualCommand : BOOL
VAR_INPUT
    Value : DINT;
END_VAR
VAR
    i : INT;
    supported : BOOL;
END_VAR
ManualCommand := FALSE;
FOR i := 1 TO CatalogCount DO
    IF Catalog[i].Value = Value THEN
        supported := TRUE;
        EXIT;
    END_IF
END_FOR
IF NOT supported THEN
    RETURN;                              // reject values outside the published set (§5.6)
END_IF
IF (_exec <> E_ExecState.READY) OR Execute OR _manualActive THEN
    RETURN;
END_IF
_manualCmd := Value;
_manualReq := TRUE;                       // consumed by the module's _M_Dispatch
_manualActive := TRUE;
Execute := TRUE;                          // rising edge enters the inherited lifecycle
ManualCommand := TRUE;
END_METHOD

// Called after the common Status mirror refresh. Derived tiers may overlay data.
METHOD PROTECTED _M_PublishStatus
;
END_METHOD

// §3.10.1 — set the module's asset identity once, at Setup. Not HMI-writable;
// identity, not configuration (deliberately outside §3.8/§7.7).
METHOD SetNameplate : BOOL
VAR_INPUT
    Plate : ST_Nameplate;
END_VAR
Nameplate := Plate;
SetNameplate := TRUE;
END_METHOD

// §3.10.2 I_ConfigSource — export the base-owned static facets this module
// deliberately keeps off the cyclic OPC UA tree. Item fragments reproduce the
// server's array naming so the HMI rebuilds the exact browse paths generically.
// A type with additional static data overrides, calls SUPER^ first, appends.
METHOD M_AppendConfig : BOOL
VAR_INPUT
    Pager : REFERENCE TO FB_ConfigPager;
END_VAR
VAR
    i    : INT;
    item : STRING(255);
END_VAR
M_AppendConfig := TRUE;
Pager.M_Append(Scope := Status.Name, Item := 'Nameplate/ProductUri',
    ValueText := Nameplate.ProductUri);
Pager.M_Append(Scope := Status.Name, Item := 'Nameplate/ManufacturerName',
    ValueText := Nameplate.ManufacturerName);
Pager.M_Append(Scope := Status.Name, Item := 'Nameplate/ProductDesignation',
    ValueText := Nameplate.ProductDesignation);
Pager.M_Append(Scope := Status.Name, Item := 'Nameplate/SerialNumber',
    ValueText := Nameplate.SerialNumber);
Pager.M_Append(Scope := Status.Name, Item := 'Nameplate/YearOfConstruction',
    ValueText := Nameplate.YearOfConstruction);
Pager.M_Append(Scope := Status.Name, Item := 'Nameplate/HardwareVersion',
    ValueText := Nameplate.HardwareVersion);
Pager.M_Append(Scope := Status.Name, Item := 'Nameplate/FirmwareVersion',
    ValueText := Nameplate.FirmwareVersion);
Pager.M_Append(Scope := Status.Name, Item := 'Nameplate/SoftwareVersion',
    ValueText := Nameplate.SoftwareVersion);
Pager.M_Append(Scope := Status.Name, Item := 'Nameplate/OrderCode',
    ValueText := Nameplate.OrderCode);
Pager.M_Append(Scope := Status.Name, Item := 'Nameplate/DocumentationUrl',
    ValueText := Nameplate.DocumentationUrl);
Pager.M_AppendNumber(Scope := Status.Name, Item := 'CatalogCount',
    Number := TO_DINT(CatalogCount));
FOR i := 1 TO CatalogCount DO
    item := CONCAT('Catalog/Catalog[', CONCAT(TO_STRING(i), ']/Value'));
    Pager.M_AppendNumber(Scope := Status.Name, Item := item, Number := Catalog[i].Value);
    item := CONCAT('Catalog/Catalog[', CONCAT(TO_STRING(i), ']/Label'));
    Pager.M_Append(Scope := Status.Name, Item := item, ValueText := Catalog[i].Label);
    // §7.6.1a - how the command is OPERATED. Without this a generic client
    // cannot tell a jog from a one-shot, and renders a hold-to-run control as a
    // click: pressing it once would latch motion nothing releases. The HMI
    // treats an absent Style as ONESHOT, so an older PLC still reads correctly.
    item := CONCAT('Catalog/Catalog[', CONCAT(TO_STRING(i), ']/Style'));
    Pager.M_AppendNumber(Scope := Status.Name, Item := item,
        Number := TO_DINT(Catalog[i].Style));
END_FOR
// §3.8b — then everything this module declared editable about itself.
_M_AppendCapabilities(Pager := Pager, Scope := Status.Name, ItemPrefix := '');
END_METHOD

// §3.8b — every value this module declared editable. The value is read live and
// the metadata comes from the same record the write will be validated against,
// so a client can never be shown a capability the PLC would not honour. Scope
// and ItemPrefix exist for the one module published under another's scope: a
// line, which a root presents as its own line data (§3.8e).
METHOD PROTECTED _M_AppendCapabilities
VAR_INPUT
    Pager      : REFERENCE TO FB_ConfigPager;
    Scope      : STRING(255);
    ItemPrefix : STRING(16);
END_VAR
VAR
    i : INT;
END_VAR
FOR i := 1 TO _nConfigWrite DO
    Pager.M_AppendCapability(Scope := Scope,
        Item := CONCAT(ItemPrefix, _pConfigWrite[i - 1].Item),
        ValueText := _M_ConfigValueText(Idx := i),
        WriteKey := _pConfigWrite[i - 1].Key,
        WriteRevision := _pConfigWrite[i - 1].Revision,
        ConfigKind := _pConfigWrite[i - 1].Kind,
        ValueType := _pConfigWrite[i - 1].ValueType,
        Writable := NOT _M_ConfigReadOnly(),
        RequiresReady := _pConfigWrite[i - 1].RequiresReady,
        HasMinimum := _pConfigWrite[i - 1].HasMinimum,
        HasMaximum := _pConfigWrite[i - 1].HasMaximum,
        Minimum := _pConfigWrite[i - 1].Minimum,
        Maximum := _pConfigWrite[i - 1].Maximum,
        Unit := _pConfigWrite[i - 1].Unit,
        LabelKey := _pConfigWrite[i - 1].LabelKey,
        EnumDomain := _pConfigWrite[i - 1].EnumDomain,
        EnumLabelKey := _pConfigWrite[i - 1].EnumLabelKey,
        ClassId := _pConfigWrite[i - 1].ClassId,
        MinReadLevel := _pConfigWrite[i - 1].MinReadLevel,
        MinWriteLevel := _pConfigWrite[i - 1].MinWriteLevel,
        ModelScoped := (_pConfigWrite[i - 1].Kind = E_ConfigKind.PAR_CFG)
            AND _M_InModelRegion(p := _pConfigWrite[i - 1].pTarget));
END_FOR
END_METHOD

// Core §3.8a - declare this module's own recipe record (its ParCfg). PAR_CFG values
// registered inside it are MODEL-SCOPED: a root can serve them for any model it
// offers, by pointing the region at that model's record for one request.
METHOD PROTECTED _M_SetModelRegion : BOOL
VAR_INPUT
    pRegion : PVOID;
    Size    : UDINT;
END_VAR
_pModelRegion := pRegion;
_modelRegionSize := Size;
_pModelView := 0;
_M_SetModelRegion := (pRegion <> 0) AND (Size > 0);
END_METHOD

METHOD PRIVATE _M_InModelRegion : BOOL
VAR_INPUT
    p : PVOID;
END_VAR
_M_InModelRegion := FALSE;
IF (_pModelRegion = 0) OR (p = 0) THEN
    RETURN;
END_IF
_M_InModelRegion := (p >= _pModelRegion) AND (p < _pModelRegion + _modelRegionSize);
END_METHOD

// Where value Idx lives for THIS request: its registered target, or - while a
// model view is open - the same offset in the viewed model's record.
METHOD PRIVATE _M_Target : PVOID
VAR_INPUT
    Idx : INT;
END_VAR
_M_Target := _pConfigWrite[Idx - 1].pTarget;
IF (_pModelView <> 0) AND (_pConfigWrite[Idx - 1].Kind = E_ConfigKind.PAR_CFG)
AND _M_InModelRegion(p := _pConfigWrite[Idx - 1].pTarget) THEN
    _M_Target := _pModelView + (_pConfigWrite[Idx - 1].pTarget - _pModelRegion);
END_IF
END_METHOD

// TRUE when WriteKey names one of this module's model-scoped values.
METHOD PROTECTED _M_ModelScopedKey : BOOL
VAR_INPUT
    WriteKey : STRING(160);
END_VAR
VAR
    i : INT;
END_VAR
_M_ModelScopedKey := FALSE;
FOR i := 1 TO _nConfigWrite DO
    IF _pConfigWrite[i - 1].Key = WriteKey THEN
        _M_ModelScopedKey := (_pConfigWrite[i - 1].Kind = E_ConfigKind.PAR_CFG)
            AND _M_InModelRegion(p := _pConfigWrite[i - 1].pTarget);
        RETURN;
    END_IF
END_FOR
END_METHOD

